            _state := 40;
        40:
            //            IF rfidInOut.stCompactModeInputMap.eResponseCode = _resetResponseCode THEN
            IF rfidInOut.xDone THEN
                THIS^.DoneWhen(TRUE);
                //                THIS^.Messenger.Info
                //                (
                //                    _stringbuilder.Append('Lock der Daten erfolgreich')
                //                        .Append('Startadresse: ')
                //                        .Append(TO_STRING(rfidinOut.udiStartAdress))
                //                        .Append(' Laenge: ')
                //                        .Append(TO_STRING(rfidInOut.uiDataLenght))
                //                        .ToString()
                //                );

                _state := 0;
            end_IF
    END_CASE
END_IF

{attribute 'monitoring' := 'call'}
PROPERTY ErrorId : RFID_FB_U.ERROR
GET
{warning disable C0371}
ErrorId := _eErrorID;
END_GET
END_PROPERTY

METHOD PUBLIC FB_init : BOOL
VAR_INPUT
    bInitRetains : BOOL; // if TRUE, the retain variables are initialized (warm start / cold start)
    bInCopyCode  : BOOL; // if TRUE, the instance afterwards gets moved into the copy code (online change)
    ParentObject : ITcoObject;
END_VAR
// This is not clear to me... I from time to time the consumer code does not see 'FB_init' of 'TcoObject', that's why overridden here with super call...
{warning disable C0316}
SUPER^.FB_init(bInitRetains, bInCopyCode, ParentObject);
END_METHOD

(*~
    <docu>
        <summary>
            Executes when task is aborted.
        </summary>
    </docu>
~*)
METHOD PROTECTED OnAbort
{warning disable C0371}
RfidInOut.eCommand := RFID_FB_U.COMMAND.IDLE;
RfidInOut.xExecute := FALSE;
RfidInOut.xAbort   := FALSE;
END_METHOD

(*~
    <docu>
        <summary>
            Executes when task reaches the ```Done``` state .
        </summary>
    </docu>
~*)
METHOD PROTECTED OnDone
{warning disable C0371}
rfidInOut.xExecute := FALSE;
rfidInOut.eCommand := RFID_FB_U.COMMAND.IDLE;
END_METHOD

(*~
    <docu>
        <summary>
            Executes when task reaches the ```Error``` state.
            <para>
                Do not confuse with <see cref="PlcDocu.TcoCore.TcoTask.WhileError()"/>, that is called cyclically until '''Error''' state is left.
            </para>
        </summary>
    </docu>
~*)
METHOD PROTECTED OnError
{warning disable C0371}
IF _noTagFound THEN
    _eErrorID := RFID_FB_U.ERROR.COMMAND_NO_TAG_FOUND;
    // not implemented by Turck
ELSIF rfidInOut.eErrorID = 16#2901 THEN
    _eErrorID := RFID_FB_U.ERROR.COMMAND_ADDRESS_OUTSIDE_BLOCK_BOUNDARIES;
ELSE
    _eErrorID := rfidInOut.eErrorID;
END_IF

THIS^.Messenger.Build().Append('Rfid Schreib/Lesekopf Fehler : ').Append(to_string(THIS^._eErrorID)).As().AsError();
END_METHOD

(*~
    <docu>
        <summary>
            Executes ones when the task starts (at the moment of transition from the ```Requested``` state into the ```Busy``` state).
        </summary>
    </docu>
~*)
METHOD PROTECTED OnStart
{warning disable C0371}
rfidInOut.eCommand := RFID_FB_U.COMMAND.IDLE;
rfidInOut.xExecute := FALSE;
rfidInOut.xAbort   := FALSE;
_state             := 10;
END_METHOD

(*~
    <docu>
        <summary>
            Restores this instance to the Ready state. Can be called explicitly or from within one of the restore mechanisms.
            <para>
                See also <see cref="PlcDocu.TcoCore.TcoTask.AutoRestorable()"/>
            </para>
        </summary>
    </docu>
~*)
METHOD Restore : ITcoRestorable
{warning disable C0371}
RfidInOut.eCommand := RFID_FB_U.COMMAND.IDLE;
RfidInOut.xExecute := FALSE;
RfidInOut.xAbort   := FALSE;
_noTagFound        := FALSE;
_eErrorID          := RFID_FB_U.ERROR.NO_ERROR;
SUPER^.Restore();
END_METHOD

END_FUNCTION_BLOCK

// ---- POUs/Turck Rfid Reader/Mock/RfidMockWorking.TcPOU
FUNCTION_BLOCK RfidMockWorking IMPLEMENTS IRfidHeadWrapper
VAR
    _timeOut        : Tc2_Standard.TON;
    _executionTimer : Tc2_Standard.TON := (PT := _executionTime);
    _executionTime  : TIME             := t#5ms;

    _udIntToMillis : UDINT := 1000;

    _resultUid : ARRAY[0..7] OF BYTE :=
    [
        16#E0
        , 16#04
        , 16#01
        , 16#50
        , 16#AC
        , 16#F4
        , 16#F3
        , 16#AD
    ];

    _states :
        (Idle
        , Busy
        , ElectedMethod
        , ReadUid
        , ReadData
        , WriteData
        , Error
        , Restore);
    _index : INT;

    _rfidInOut : RfidInOut;
END_VAR

{warning disable C0371}
//28 blocks, 4 bytes each, => 112 bytes max user Memory!

CASE _states OF
    Idle:
        _rfidInOut.xbusy := _rfidInOut.xExecute;
        _rfidInOut.xTP   := TRUE;

        IF _rfidInOut.xbusy THEN
            _states := Busy;
        END_IF

    Busy:

        _rfidInOut.uiDataRxLength := _rfidInOut.uiDataLenght;
        _timeOut(in := _rfidInOut.xbusy, PT := UDINT_TO_TIME(_rfidInOut.udiTimeOut) / _udintToMillis);
        _executionTimer(in := _rfidInOut.xBusy);

        IF _timeOut.Q THEN
            _states             := Error;
            _rfidInOut.eErrorID := RFID_FB_U.ERROR.TIME_OUT;
            RETURN;

        ELSIF _executionTimer.Q THEN
            _states := ElectedMethod;
        END_IF

    ElectedMethod:
        IF _rfidInOut.uiDataLenght > 112 THEN
            _states             := Error;
            _rfidInOut.eErrorID := RFID_FB_U.ERROR.COMMAND_LENGTH_OUTSIDE_TAG_SPECS;
            RETURN;
        ELSIF _rfidInOut.udiStartAdress > 112 THEN
            _states             := Error;
            _rfidInOut.eErrorID := RFID_FB_U.ERROR.COMMAND_ADDRESS_OUTSIDE_TAG_SPECS;
            RETURN;
        END_IF

        IF _rfidInOut.eCommand = RFID_FB_U.COMMAND.INVENTORY THEN
            FOR _index := 0 TO 7 DO
                _rfidInOut.myReadData[_index] := _resultUid[_index];
            END_FOR

            _rfidInOut.xbusy := FALSE;
            _rfidInOut.xDone := TRUE;
        ELSIF _rfidInOut.eCommand = RFID_FB_U.COMMAND.READ THEN

            FOR _index := 0 TO UINT_TO_INT(_rfidInOut.uiDataLenght) - 1 DO
                _rfidInOut.myReadData[_index] := 16#05 + INT_TO_BYTE(_index + UDINT_TO_INT(_rfidInOut.udiStartAdress));
            END_FOR

            _rfidInOut.xbusy := FALSE;
            _rfidInOut.xDone := TRUE; //

        ELSIF _rfidInOut.eCommand = RFID_FB_U.COMMAND.WRITE THEN
            _rfidInOut.xbusy := FALSE;
            _rfidInOut.xDone := TRUE;

        ELSIF _rfidInOut.eCommand = RFID_FB_U.COMMAND.SET_PERMA_LOCK THEN
            _rfidInOut.xbusy := FALSE;
            _rfidInOut.xDone := TRUE;
        END_IF

    Error:
        _executionTimer(in := FALSE);
        _timeOut(in := FALSE);
        _rfidInOut.xbusy  := FALSE;
        _rfidInOut.xError := TRUE;

        IF NOT _rfidInOut.xExecute THEN
            _States := Restore;
        END_IF
    Restore:
        _rfidInOut.xDone    := FALSE;
        _rfidInOut.xError   := FALSE;
        _rfidInOut.eErrorID := RFID_FB_U.ERROR.NO_ERROR;
        _States             := Idle;
END_CASE

METHOD Execute
VAR_INPUT
    xExecute       : BOOL;
    xAbort         : BOOL;
    udiTimeOut     : UDINT := 10000;
    eCommand       : RFID_FB_U.COMMAND;
    udiStartAdress : UDINT;
    uiDataLenght   : UINT;
    myWriteData    : ARRAY[0..127] OF BYTE;
END_VAR
VAR_OUTPUT
    myReadData          : ARRAY[0..127] OF BYTE;
    xDone               : BOOL;
    xBusy               : BOOL;
    xError              : BOOL;
    xAborted            : BOOL;
    eErrorID            : RFID_FB_U.ERROR;
    xTP                 : BOOL;
    xRWHeadNotCOnnected : BOOL;
    uiDataRxLength      : UINT;
END_VAR
VAR_INST
    _busy : BOOL;
END_VAR
THIS^();

_rfidInOut.xExecute       := xExecute;
_rfidInOut.xAbort         := xAbort;
_rfidInOut.udiTimeOut     := udiTimeOut;
_rfidInOut.eCommand       := eCommand;
_rfidInOut.udiStartAdress := udiStartAdress;
_rfidInOut.uiDataLenght   := uiDataLenght;
_rfidInOut.myWriteData    := myWriteData;

myReadData          := _rfidInOut.myReadData;
xDone               := _rfidInOut.xDone;
xBusy               := _rfidInOut.xBusy;
xError              := _rfidInOut.xError;
xAborted            := _rfidInOut.xAborted;
eErrorID            := _rfidInOut.eErrorID;
xTP                 := _rfidInOut.xTP;
xRWHeadNotCOnnected := _rfidInOut.xRWHeadNotCOnnected;
uiDataRxLength      := _rfidInOut.uiDataRxLength;
END_METHOD

END_FUNCTION_BLOCK

// ---- Test/Engel Ethercat Bridge Comm Tests/EngelInput_Test.TcPOU
FUNCTION_BLOCK EngelInput_Test EXTENDS TcUnit.FB_TestSuite
VAR

END_VAR

ParseVariantOne();

METHOD PRIVATE ParseVariantOne
VAR_INST
    in : ARRAY[1..42] OF BYTE;

    engelInput : EngelInput;

    inputData : EngelInputData;
END_VAR
// lebenssignal: alle 6ms muss der Zaehler um 1 erhoet werden (0-255, 0-255)
// will be the Counter be incremented from me and engel,
// will there be 2 Counter, everybody responsible for his
// what is the Result, if not incremented

//

Test('ParseVariantOne');

in[1]  := 255;
in[2]  := 255;
in[39] := 2#1111_1111;

engelInput(input := in);

inputData := engelInput.GetInputData();

AssertEquals_UINT(Expected := 65535, Actual := inputData.HeartBeat, 'Heartbeat not Correct');
AssertTrue(Condition := inputData.AutoActive, ' AutomatikActive should be true');
AssertTrue(Condition := inputData.HomeDone, 'HomeDoneshould be true');
AssertTrue(Condition := inputData.ManualActive, 'ManualActive should be true');
AssertTrue(Condition := inputData.HomeRequest, 'RequestHome should be true');
AssertTrue(Condition := inputData.SafetyClosed, 'SafetyClosed should be true');
AssertTrue(Condition := inputData.SafetyOpeningAllowed, 'SafetyOpeningAllowed should be true');
AssertTrue(Condition := inputData.AutoStart, 'StartAuto should be true');

TEST_FINISHED();
END_METHOD

END_FUNCTION_BLOCK

// ---- POUs/Engel Ethercat Bridge Communication/FunctionBlocks/EngelInput.TcPOU
FUNCTION_BLOCK EngelInput IMPLEMENTS IInput
VAR_INPUT
    input : ARRAY[1..42] OF BYTE;
END_VAR

METHOD GetInputData : EngelInputData
VAR
    hbTemp : uint;
END_VAR
hbTemp := input[1];
hbTemp := SHL(hbTemp, 8);
hbTemp := hbTemp OR input[2];

GetInputData.HeartBeat            := hbTemp;
GetInputData.ManualActive         := input[39].0;
GetInputData.AutoActive           := input[39].1;
GetInputData.AutoStart            := input[39].2;
GetInputData.HomeRequest          := input[39].3;
GetInputData.HomeDone             := input[39].4;
GetInputData.SafetyClosed         := input[39].5;
GetInputData.SafetyOpeningAllowed := input[39].6;
END_METHOD

END_FUNCTION_BLOCK

// ---- POUs/Engel Ethercat Bridge Communication/FunctionBlocks/HeartBeat.TcPOU
FUNCTION_BLOCK HeartBeat IMPLEMENTS IHeartBeat
VAR_INPUT
    execute : BOOL;
END_VAR

VAR
    heartBeatTimer : TON;
    eState         : eHeartBeatState;
    erroString     : T_MaxString;
    heartBeat      : UINT;

END_VAR

IF execute THEN
    heartBeatTimer();

    CASE eState OF
        eHeartBeatState.Unknown:
            CheckStates();
        eHeartBeatState.Valid:
            heartBeatTimer(in := TRUE);
            erroString := '';
            CheckStates();
        eHeartBeatState.Timeout:
            erroString := CONCAT
            (
                'Timeout, da keine Erhoehung Heartbeat stattgefunden hat in '
                , TO_STRING(GetHeartBeatTimeOutTime)
            );
    ELSE
        ;
    END_CASE
END_IF

METHOD PRIVATE CheckStates : BOOL
VAR_INPUT
END_VAR
IF execute THEN
    IF heartBeatTimer.Q THEN
        SetState(eHeartBeatState.Timeout);
    END_IF
ELSE
    SetState(eHeartBeatState.Unknown);
END_IF
END_METHOD

METHOD FB_init : BOOL
VAR_INPUT
    bInitRetains         : BOOL; // if TRUE, the retain variables are initialized (warm start / cold start)
    bInCopyCode          : BOOL; // if TRUE, the instance afterwards gets moved into the copy code (online change)
    heartBeatTimeoutTime : TIME;
END_VAR
heartBeatTimer.PT := heartBeatTimeoutTime;

this^.eState := eHeartBeatState.Unknown;
END_METHOD

PROPERTY GetErrorMessage : T_MaxString;
GET
GetErrorMessage := erroString;
END_GET
END_PROPERTY

//actual Heartbeat of PLC
PROPERTY GetHeartBeat : UINT
GET
IF NOT execute THEN
    THIS^.erroString := 'Bitte Execute auf True setzten!';
    RETURN;
END_IF

GetHeartBeat := heartBeat;
END_GET
END_PROPERTY

PROPERTY GetHeartbeatTimeoutTime : TIME
GET
GetHeartbeatTimeoutTime := heartBeatTimer.PT;
END_GET
END_PROPERTY

PROPERTY GetState : eHeartBeatState
GET
GetState := eState;
END_GET
END_PROPERTY

// Increases HB +1 from InputValue
METHOD IncreaseHeartBeat : UINT
VAR_INPUT
    externalHeartBeat : UINT;
END_VAR
IF NOT execute THEN
    THIS^.erroString  := 'Bitte Execute auf True setzten!';
    IncreaseHeartBeat := 0;
    RETURN;
END_IF

SetState(eHeartBeatState.Valid);
ResetTimer();

IF externalHeartBeat >= 255 THEN
    IncreaseHeartBeat := 0;
ELSE
    IncreaseHeartBeat := externalHeartBeat + 1;
END_IF

heartBeat := IncreaseHeartBeat;
END_METHOD

METHOD PRIVATE ResetTimer
VAR_INPUT
END_VAR
THIS^.heartBeatTimer(IN := false);
END_METHOD

METHOD PRIVATE SetState
VAR_INPUT
    eState : eHeartBeatState;
END_VAR
This^.eState := eState;
END_METHOD

END_FUNCTION_BLOCK

// ---- Test/Engel Ethercat Bridge Comm Tests/EngelOutput_Test.TcPOU
FUNCTION_BLOCK EngelOutput_Test EXTENDS FB_TestSuite

SetOutputsAndVerify();

METHOD PRIVATE SetOutputsAndVerify
VAR
    out : EngelOutput;
END_VAR
TEST('SetOutputsAndVerify');

out.ManualActive(TRUE);
AssertEquals_BYTE(Expected := 2#0000_0001, Actual := out.output[39], 'SetManualActive is true');
out.ManualActive(FALSE);

out.AutomaticIsActive(TRUE);
AssertEquals_BYTE(Expected := 2#0000_0010, Actual := out.output[39], 'SetAutomaticeActive is true');
out.AutomaticIsActive(FALSE);

out.StartAutomatic(TRUE);
AssertEquals_BYTE(Expected := 2#0000_0100, Actual := out.output[39], 'SetStart is true');
out.StartAutomatic(FALSE);

out.RequestHome(TRUE);
AssertEquals_BYTE(Expected := 2#0000_1000, Actual := out.output[39], 'SetRequestHome is true');
out.RequestHome(FALSE);

out.HomeIsDone(TRUE);
AssertEquals_BYTE(Expected := 2#0001_0000, Actual := out.output[39], 'SetHomeDone is true');
out.HomeIsDone(FALSE);

out.SafetyIsClosed(TRUE);
AssertEquals_BYTE(Expected := 2#0010_0000, Actual := out.output[39], 'SetSafetyClosed is true');
out.SafetyIsClosed(FALSE);

out.RequestSafetyOpening(TRUE);
AssertEquals_BYTE(Expected := 2#0100_0000, Actual := out.output[39], 'SetSafetyOpeningRequest is true');
out.RequestSafetyOpening(FALSE);

out.SetHeartBeat(65535);
AssertEquals_BYTE(Expected := 255, Actual := out.output[1], 'Byte  1 Heartbeat shall be 255');
AssertEquals_BYTE(Expected := 255, Actual := out.output[2], 'Byte  2 Heartbeat shall be 255');

TEST_FINISHED();
END_METHOD

END_FUNCTION_BLOCK

// ---- POUs/Engel Ethercat Bridge Communication/FunctionBlocks/EngelOutput.TcPOU
FUNCTION_BLOCK EngelOutput IMPLEMENTS IOutput
VAR_OUTPUT
    output : ARRAY[0..42] OF BYTE;
END_VAR

METHOD PUBLIC AutomaticIsActive
VAR_INPUT
    enable : BOOL;
END_VAR

output[39].1 := enable;
END_METHOD

METHOD PUBLIC HomeIsDone
VAR_INPUT
    enable : BOOL;
END_VAR
output[39].4 := enable;
END_METHOD

METHOD PUBLIC ManualActive
VAR_INPUT
    enable : BOOL;
END_VAR
output[39].0 := enable;
END_METHOD

METHOD PUBLIC RequestHome
VAR_INPUT
    enable : BOOL;
END_VAR
output[39].3 := enable;
END_METHOD

METHOD PUBLIC RequestSafetyOpening
VAR_INPUT
    enable : BOOL;
END_VAR
output[39].6 := enable;
END_METHOD

METHOD PUBLIC SafetyIsClosed
VAR_INPUT
    enable : BOOL;
END_VAR
output[39].5 := enable;
END_METHOD

METHOD SetHeartBeat
VAR_INPUT
    heartBeat : UINT;
END_VAR
output[1].0 := heartBeat.0;
output[1].1 := heartBeat.1;
output[1].2 := heartBeat.2;
output[1].3 := heartBeat.3;
output[1].4 := heartBeat.4;
output[1].5 := heartBeat.5;
output[1].6 := heartBeat.6;
output[1].7 := heartBeat.7;

output[2].0 := heartBeat.8;
output[2].1 := heartBeat.9;
output[2].2 := heartBeat.10;
output[2].3 := heartBeat.11;
output[2].4 := heartBeat.12;
output[2].5 := heartBeat.13;
output[2].6 := heartBeat.14;
output[2].7 := heartBeat.15;
END_METHOD

METHOD PUBLIC StartAutomatic
VAR_INPUT
    enable : BOOL;
END_VAR
output[39].2 := enable;
END_METHOD

END_FUNCTION_BLOCK

// ---- Test/Engel Ethercat Bridge Comm Tests/HeartBeat_Test.TcPOU
FUNCTION_BLOCK HeartBeat_Test EXTENDS TcUnit.FB_TestSuite

GetsValueAndGiveBackIncreasedValueStatusValid();
HeartbeatFromEngelTimeout_GetStateGivesStatusTimeOut();
ErrorOccurs_ExpectStringMessage();
AfterTimeOutRecieveNewHb_ExpectToChangeStatusBackToValid();
NotExecute_ExpectErrorMessageAndStateUnknown();

METHOD PRIVATE AfterTimeOutRecieveNewHb_ExpectToChangeStatusBackToValid
VAR_INST
    toTimer : TON := (PT := T#4MS); // Bigger 12ms !
    eState  : eHeartBeatState;
    first   : BOOL := TRUE;
    hb      : HeartBeat(heartBeatTimeoutTime := T#2MS);
    resetHb : BOOL;

END_VAR
Test('ErrorOccurs_ExpectStringAfterTimeOutRecieveNewHb_ExpectToChangeStatusBackToValidMessage');
// Arrange
// Act
// Assert
hb(execute := TRUE);
toTimer();

IF first THEN
    first  := FALSE;
    eState := hb.GetState;
    hb.IncreaseHeartBeat(5);
    eState := hb.GetState;
    AssertEquals_UINT(6, hb.GetHeartBeat, 'Nach Erhoehung muss HB 6 sein');
    AssertTrue(eState = eHeartBeatState.Valid, 'State muss Valid sein');
    toTimer(in := TRUE);
END_IF

IF toTimer.q THEN
    AssertTrue(hb.GetState = eHeartBeatState.Timeout, 'Timeout, keine Erhoehung HB durch Engel');
    resetHb := TRUE;
END_IF

IF resetHb THEN
    hb.IncreaseHeartBeat(665);
    AssertTrue(hb.GetState = eHeartBeatState.Valid, 'State muss Valid sein');
    AssertEquals_UINT(0, hb.GetHeartBeat, 'Nach Erhoehung muss HB 0 sein');

    TEST_FINISHED();
END_IF
END_METHOD

METHOD PRIVATE ErrorOccurs_ExpectStringMessage
VAR_INST
    hb                 : HeartBeat(heartBeatTimeoutTime := T#1MS);
    toTimer            : TON := (PT := T#3MS); // Bigger 12ms !
    errorMessage       : STRING;
    actualErrorMessage : STRING;
    first              : BOOL := TRUE;
    eState             : eHeartBeatState;

END_VAR
Test('ErrorOccurs_ExpectStringMessage');
// Arrange
// Act
// Assert

hb(execute := TRUE);
toTimer(in := TRUE);

IF first THEN
    errorMessage       := '';
    actualErrorMessage := hb.GetErrorMessage;
    AssertEquals_STRING(errorMessage, actualErrorMessage, 'ErrorMessage soll leer sein');
    first := FALSE;
    hb.IncreaseHeartBeat(1);
END_IF

IF toTimer.Q THEN
    eState := hb.GetState;
    AssertTrue(eState = eHeartBeatState.Timeout, 'Timeout, keine Erhoehung HB durch Engel');
    actualErrorMessage := hb.GetErrorMessage;

    errorMessage := CONCAT
    (
        'Timeout, da keine Erhoehung Heartbeat stattgefunden hat in '
        , TO_STRING(hb.GetHeartBeatTimeOutTime)
    );

    AssertEquals_STRING(errorMessage, actualErrorMessage, 'ErrorMessage muss gleich sein');

    TEST_FINISHED();
end_if
END_METHOD

METHOD PRIVATE GetsValueAndGiveBackIncreasedValueStatusValid
VAR
    hb            : HeartBeat(heartBeatTimeoutTime := T#12MS);
    eState        : eHeartBeatState;
    inputData     : UINT;
    inHeartBeat   : UINT := 0;
    expectedOutHb : UINT := 1;
END_VAR
// Calculate a Heartbeat for the Engle Ethercat Bridge Communication
// Wertebereich des Heartbeats ist [0..65635]
// Aber Engel erhoeht internen Zaehler alle 6ms bis 255!
// Nur Aenderung von meiner Seite notwendig
// Wenn nach max. 12ms keine Aenderung => Fehler

Test('GetsValueAndGiveBackIncreasedValueStatusValid');
// Arrange
// Act
// Assert

hb(execute := TRUE);

eState := hb.GetState;
AssertTrue(estate = eHeartBeatState.Unknown, 'State soll Unknown sein');
///=========================================================

inputData := hb.IncreaseHeartBeat(inHeartBeat);
eState    := hb.GetState;
AssertEquals_UINT(expectedOutHb, inputData, 'Nach Erhoehung muss HB 1 sein');
AssertTrue(estate = eHeartBeatState.Valid, 'State muss Valid sein');

//Arrange
inHeartBeat   := 255;
expectedOutHb := 0;

//Act
inputData := hb.IncreaseHeartBeat(inHeartBeat);
AssertEquals_UINT(expectedOutHb, inputData, 'Nach Erhoehung ueber 255 muss HB wieder 0 sein');
AssertTrue(estate = eHeartBeatState.Valid, 'State muss Valid sein');

TEST_FINISHED();
END_METHOD

METHOD PRIVATE HeartbeatFromEngelTimeout_GetStateGivesStatusTimeOut
VAR
    inputData     : UINT;
    inHeartBeat   : UINT := 22;
    expectedOutHb : UINT := 23;
END_VAR

VAR_INST
    toTimer : TON := (PT := T#20MS); // Bigger 12ms !
    eState  : eHeartBeatState;
    first   : BOOL := TRUE;
    hb      : HeartBeat(heartBeatTimeoutTime := T#12MS);

END_VAR
// Calculate a Heartbeat for the Engle Ethercat Bridge Communication
// Wertebereich des Heartbeats ist [0..65635]
// Aber Engel erhoeht internen Zaehler alle 6ms bis 255!
// Nur Aenderung von meiner Seite notwendig
// Wenn nach max. 12ms keine Aenderung => Fehler

Test('HeartbeatFromEngelTimeout_GetStateGivesStatusTimeOut');
// Arrange
// Act
// Assert
hb(execute := TRUE);
toTimer();

IF first THEN
    first  := FALSE;
    eState := hb.GetState;
    AssertTrue(estate = eHeartBeatState.Unknown, 'State soll Unknown sein');
    ///=========================================================

    inputData := hb.IncreaseHeartBeat(inHeartBeat);
    eState    := hb.GetState;
    AssertEquals_UINT(expectedOutHb, inputData, 'Nach Erhoehung muss HB 23 sein');
    AssertEquals_UINT(expectedOutHb, hb.GetHeartBeat, 'Bie GetHeartBeat muss HB 23 sein');
    AssertTrue(estate = eHeartBeatState.Valid, 'State muss Valid sein');
    //======================

    toTimer(in := TRUE);
END_IF

IF toTimer.ET <= T#12MS THEN
    AssertTrue(estate = eHeartBeatState.Valid, 'Valid, TO erst nach 12ms');
END_IF

IF toTimer.Q THEN
    eState := hb.GetState;
    AssertTrue(estate = eState, 'Timeout, keine Erhoehung HB durch Engel');
    TEST_FINISHED();
END_IF
END_METHOD

METHOD PRIVATE NotExecute_ExpectErrorMessageAndStateUnknown
VAR
    timeout             : TIME := T#1MS;
    hb                  : HeartBeat(heartBeatTimeoutTime := timeout);
    errorStringExpected : STRING;
    errorStringActual   : STRING;
END_VAR
TEST('NotExecute_ExpectErrorMessageAndStateUnknown');

hb(execute := FALSE);
hb.IncreaseHeartBeat(23);
errorStringExpected := 'Bitte Execute auf True setzten!';
errorStringActual   := hb.GetErrorMessage;
AssertEquals_STRING(errorStringActual, errorStringExpected, 'ErrorMessage soll gleich sein');
AssertTrue(hb.GetState = eHeartBeatState.Unknown, 'State muss Unknown sein');
AssertEquals_UINT(hb.IncreaseHeartBeat(25), 0, 'Keine Erhoehung, da Execute False');
AssertEquals_UINT(hb.GetHeartBeat, 0, 'Keine Erhoehung, da Execute False');
AssertTrue(hb.GetHeartbeatTimeoutTime = timeout, 'Property muss gleiche Zeit wie bei Init zurueckgeben (1ms)');

TEST_FINISHED();
END_METHOD

END_FUNCTION_BLOCK

// ---- Test/Sequences/Test/SequenceTryout_Test.TcPOU
FUNCTION_BLOCK SequenceTryout_Test EXTENDS TcUnit.FB_TestSuite IMPLEMENTS TcoCore.ITcoContext
VAR
    //Context for TcOpen
    _nfContext : TcoCore.TcoContextNfCompatibility;
END_VAR

VAR
    //~
    autoSequenceTryOutTest : SequenceTryout(THIS^, eRestoreMode.AutoRestoreMembers);
    //~
END_VAR


_nfContext.VolatileOpen(); //Required for TCopen
//==============================================
GivenThatEverythingWorksExpectCompleteSequenceToFinishInDone();
//==============================================
_nfContext.VolatileClose();

PROPERTY Context : TcoCore.ITcoContext
GET
Context := This^._nfContext;
END_GET
END_PROPERTY

PROPERTY EndCycleCount : ULINT
GET
EndCycleCount := THIS^._nfContext._endCycleCount;
END_GET
END_PROPERTY

PROPERTY Environment : TcoCore.ITcoContextEnvironment
GET
Environment := THIS^._nfContext._settings;
END_GET
END_PROPERTY

METHOD PRIVATE GivenThatEverythingWorksExpectCompleteSequenceToFinishInDone

VAR
    state                : INT;
    context              : ITcoContext;
    autoRestorable       : BOOL;
    currentStep          : StepDetails;
    euqalsTo             : BOOL;
    identity             : ULINT;
    isAutoRestoreEnabled : BOOL;
    isFreshState         : BOOL;
    lastStateChangeCycle : ULINT;
    messenger            : ITcoMessenger;
    modeController       : ITcoSequencerModeController;
    observer             : ITcoSequencerObserver;
    parent               : ITcoObject;

END_VAR

VAR
    currentStepActive : StepDetails;
END_VAR
//{warning disable C0371}
TcUnit.TEST('GivenThatEverythingWorksExpectCompleteSequenceToFinishInDone');
//Arrange

//autoSequenceTryOutTest.Restore();
currentStepActive.ID := 0;

////Act
autoSequenceTryOutTest.Run();

////Assert

//AssertEquals(Expected := currentStepActive.ID, Actual := autoSequenceTryOutTest.CurrentStep.ID, Message := 'Muss Step 999 sein');

state                := autoSequenceTryOutTest.State;
context              := autoSequenceTryOutTest.Context;
autorestorable       := autoSequenceTryOutTest.AutoRestorable;
currentStep          := autoSequenceTryOutTest.CurrentStep;
Identity             := autoSequenceTryOutTest.Identity;
isAutoRestoreEnabled := autoSequenceTryOutTest.IsAutoRestoreEnabled;
isFreshState         := autoSequenceTryOutTest.IsFreshState;
LastStateChangeCycle := autoSequenceTryOutTest.LastStateChangeCycle;
messenger            := autoSequenceTryOutTest.Messenger;
ModeController       := autoSequenceTryOutTest.ModeController;
Observer             := autoSequenceTryOutTest.Observer;
Parent               := autoSequenceTryOutTest.Parent;

IF (autoSequenceTryOutTest.CurrentStep.Duration >= T#10MS) OR autoSequenceTryOutTest.State = 999 THEN
    //autoSequenceTryOutTest.Restore();
    currentStepActive.ID := 999;
    AssertEquals
    (
        Expected  := currentStepActive.ID
        , Actual  := autoSequenceTryOutTest.CurrentStep.ID
        , Message := 'Muss Step 999 sein'
    );

    TcUnit.TEST_FINISHED();
END_IF
END_METHOD

PROPERTY Identity : ULINT
GET
Identity := THIS^._nfContext._Identity;
END_GET
END_PROPERTY

PROPERTY Logger : TcoCore.ITcoLogger
GET
Logger := THIS^._nfContext._logger;
END_GET
END_PROPERTY

PROPERTY RealTimeClock : TcoCore.ITcoRtc
GET
RealTimeClock := THIS^._nfContext._rtc;
END_GET
END_PROPERTY

PROPERTY StartCycleCount : ULINT
GET
StartCycleCount := THIS^._nfContext._startCycleCount;
END_GET
END_PROPERTY

END_FUNCTION_BLOCK

// ---- POUs/Sequences/Test/SequenceTryout.TcPOU
FUNCTION_BLOCK SequenceTryout EXTENDS TcoCore.TcoSequencer
VAR
    counter : INT;
END_VAR
VAR
    //    eSequenceTest : E_SequenceTest := E_SequenceTest.WaitForStart;
    eSequenceTest : stSequenceTest;
    itfValveA     : I_DualPositionActuator := valveA;
    //~
    valveA : FB_DualPositionActuator
    (
        tActivateTimeout                     := T#3S
        , tDisableTimeout                    := T#3S
        , bIsActiveFeedbackSensorAvailable   := TRUE
        , bIsDisabledFeedbackSensorAvailable := TRUE
        , bNormallyDisabled                  := TRUE
    );
    //~
END_VAR
VAR CONSTANT
    simV : INT := 4;
END_VAR

(*~
    <docu>
        <summary>
            Main method of the sequener. Custom code needs to be placed here. The sequencer is executed by call of InstanceName.Run() method.
            This method is abstract, and it must be overridden in derived block.
        </summary>
    </docu>
~*)
METHOD PROTECTED Main : BOOL
counter := counter + 1;

IF (Step(eSequenceTest.WaitForStart, TRUE, 'Restore und Start')) THEN
    //    eSequenceTest := stSequenceTest.OpenValveAandB;
    StepCompleteWhen(counter MOD simV = 0);
END_IF

IF (Step(eSequenceTest.OpenValveAandB, TRUE, 'Zweiter Step')) THEN
    StepCompleteWhen(counter MOD simV = 0);
END_IF

IF (Step(999, TRUE, 'SEQUENCE COMPLETE')) THEN
    //--------------------------------------------
    CompleteSequence();
    //--------------------------------------------
END_IF;

IF (step(909, TRUE, 'ERROR Handling')) THEN
    ;
END_IF
END_METHOD

(*~
    <docu>
        <summary>
            This method is executed upon step completion.
            This method can be overridden in derived block by custom logic.
        </summary>
    </docu>
~*)
METHOD PROTECTED OnStepCompleted
counter := 1;
END_METHOD

END_FUNCTION_BLOCK

// ---- POUs/Counter Allgemein/Counter.TcPOU
//{attribute 'hide_all_locals'}
FUNCTION_BLOCK Counter EXTENDS TcoCore.TcoObject IMPLEMENTS ICounter
VAR
    _countStep  : UDINT;
    _countValue : UDINT;
    _countLimit : UDINT;

END_VAR

METHOD CountDown
_countValue := _countValue - _countStep;
END_METHOD

{attribute 'monitoring' := 'variable'}
PROPERTY CountLimitReached : BOOL
GET
CountLimitReached := CountValue >= _countLimit;
END_GET
END_PROPERTY

METHOD CountUp

_countValue := _countValue + _countStep;
END_METHOD

{attribute 'monitoring' := 'monitor'}
PROPERTY CountValue : UDINT
GET
CountValue := _countValue;
END_GET
END_PROPERTY

{attribute 'monitoring' := 'variable'}
PROPERTY CountZeroReached : BOOL
GET
CountZeroReached:= CountValue = 0;
END_GET
END_PROPERTY

{attribute 'hide'}
METHOD FB_init : BOOL
VAR_INPUT
    (* if TRUE, the retain variables are initialized (warm start / cold start)*)
    bInitRetains : BOOL;
    (* if TRUE, the instance afterwards gets moved into the copy code (online change)*)
    bInCopyCode  : BOOL;
    ParentObject : ITcoObject;

    countStep      : UDINT;
    countInitValue : UDINT;
    countLimit     : UDINT;
END_VAR
//SUPER^.FB_init(bInitRetains, bInCopyCode, ParentObject);

_countStep := countStep;
_countValue := countInitValue;
_countLimit := countLimit;

IF countInitValue > countLimit THEN
    Messenger.Error('Value groesser als Limit eingestellt');
    RETURN;
END_IF
END_METHOD

METHOD ResetCount
_countValue := 0;
END_METHOD

END_FUNCTION_BLOCK

// ---- POUs/DualPositionActuator/POUs/FB_DualPositionActuator.TcPOU
FUNCTION_BLOCK FB_DualPositionActuator IMPLEMENTS I_DualPositionActuator
VAR
    {attribute 'TcHmiSymbol.Show'}
    {attribute 'TcHmiSymbol.ReadOnly'}
    eState                             : E_DualPositionActuatorState;
    fbTimerActivatingTimeout           : TON;
    fbTimerDisablingTimeout            : TON;
    bIsActiveFeedbackSensorAvailable   : BOOL;
    bIsDisabledFeedbackSensorAvailable : BOOL;

    bIsNormallyDisabled : BOOL; // [True = Normally disabled, False = Normally activated]
END_VAR
VAR_INPUT
    bActiveFeedback  : BOOL; // Sensor input
    bDisableFeedback : BOOL; // Sensor input
END_VAR
VAR_OUTPUT
    bActivate : BOOL; // Actuator output
    bDisable  : BOOL; // Actuator output
END_VAR

CASE eState OF
    E_DualPositionActuatorState.Unknown:
        CheckFeedback();

    E_DualPositionActuatorState.Active:
        CheckFeedback();

    E_DualPositionActuatorState.Disabled:
        CheckFeedback();

    E_DualPositionActuatorState.TimeoutActivating:
        IF bIsNormallyDisabled THEN
            bActivate := FALSE;
        ELSE
            CheckFeedback();
        END_IF

    E_DualPositionActuatorState.TimeoutDisabling:
        IF NOT bIsNormallyDisabled THEN
            bDisable := FALSE;
        ELSE
            CheckFeedback();
        END_IF

    E_DualPositionActuatorState.Activating:
        IF NOT bIsActiveFeedbackSensorAvailable AND NOT bIsDisabledFeedbackSensorAvailable THEN
            SetState(eState := E_DualPositionActuatorState.Active);
        ELSIF NOT bIsActiveFeedbackSensorAvailable AND NOT bDisableFeedback THEN
            SetState(eState := E_DualPositionActuatorState.Active);
        ELSIF NOT bIsActiveFeedbackSensorAvailable AND bDisableFeedback THEN
            fbTimerActivatingTimeout(IN := TRUE);

            IF fbTimerActivatingTimeout.Q THEN
                SetState(eState := E_DualPositionActuatorState.TimeoutActivating);
            END_IF
        ELSE
            fbTimerActivatingTimeout(IN := TRUE);

            IF fbTimerActivatingTimeout.Q THEN
                SetState(eState := E_DualPositionActuatorState.TimeoutActivating);
            END_IF

            CheckFeedback();
        END_IF

    E_DualPositionActuatorState.Disabling:
        IF NOT bIsDisabledFeedbackSensorAvailable AND NOT bIsActiveFeedbackSensorAvailable THEN
            SetState(eState := E_DualPositionActuatorState.Disabled);
        ELSIF NOT bIsDisabledFeedbackSensorAvailable AND NOT bActiveFeedback THEN
            SetState(eState := E_DualPositionActuatorState.Disabled);
        ELSIF NOT bIsDisabledFeedbackSensorAvailable AND bActiveFeedback THEN
            fbTimerDisablingTimeout(IN := TRUE);

            IF fbTimerDisablingTimeout.Q THEN
                SetState(eState := E_DualPositionActuatorState.TimeoutDisabling);
            END_IF
        ELSE
            fbTimerDisablingTimeout(IN := TRUE);

            IF fbTimerDisablingTimeout.Q THEN
                SetState(eState := E_DualPositionActuatorState.TimeoutDisabling);
            END_IF

            CheckFeedback();
        END_IF
END_CASE

METHOD PUBLIC Activate
IF GetState() = E_DualPositionActuatorState.Activating OR GetState() = E_DualPositionActuatorState.Active THEN
    RETURN;
END_IF

SetState(eState := E_DualPositionActuatorState.Activating);
fbTimerActivatingTimeout(IN := FALSE);
bDisable  := FALSE;
bActivate := TRUE;
END_METHOD

METHOD PRIVATE CheckFeedback
IF eState = E_DualPositionActuatorState.TimeoutActivating OR eState = E_DualPositionActuatorState.TimeoutDisabling THEN
    RETURN;
ELSIF bActiveFeedback AND NOT bDisableFeedback AND eState <> E_DualPositionActuatorState.Disabling THEN
    SetState(eState := E_DualPositionActuatorState.Active);
ELSIF bDisableFeedback AND NOT bActiveFeedback AND eState <> E_DualPositionActuatorState.Activating THEN
    SetState(eState := E_DualPositionActuatorState.Disabled);
ELSIF NOT bActiveFeedback
          AND bIsActiveFeedbackSensorAvailable
          AND NOT bIsDisabledFeedbackSensorAvailable
          AND eState <> E_DualPositionActuatorState.Activating THEN
    SetState(eState := E_DualPositionActuatorState.Disabled);
ELSIF NOT bDisableFeedback
          AND bIsDisabledFeedbackSensorAvailable
          AND NOT bIsActiveFeedbackSensorAvailable
          AND eState <> E_DualPositionActuatorState.Disabling THEN
    SetState(eState := E_DualPositionActuatorState.Active);
ELSIF bActiveFeedback AND bDisableFeedback THEN
    SetState(eState := E_DualPositionActuatorState.Unknown);
END_IF
END_METHOD

METHOD PUBLIC Disable
IF GetState() = E_DualPositionActuatorState.Disabling OR GetState() = E_DualPositionActuatorState.Disabled THEN
    RETURN;
END_IF

SetState(eState := E_DualPositionActuatorState.Disabling);
fbTimerDisablingTimeout(IN := FALSE);
bDisable  := TRUE;
bActivate := FALSE;
END_METHOD

METHOD FB_init : BOOL
VAR_INPUT
    bInitRetains     : BOOL; // if TRUE, the retain variables are initialized (warm start / cold start)
    bInCopyCode      : BOOL; // if TRUE, the instance afterwards gets moved into the copy code (online change)
    tActivateTimeout : TIME;
    tDisableTimeout  : TIME;
    bIsActiveFeedbackSensorAvailable
        : BOOL;                                // Set this to true if feedback is provided by a sensor
    bIsDisabledFeedbackSensorAvailable : BOOL; // Set this to true if feedback is provided by a sensor
    bNormallyDisabled                  : BOOL; // [True = Normally disabled, False = Normally activated]
END_VAR
fbTimerActivatingTimeout.PT := tActivateTimeout;
fbTimerDisablingTimeout.PT  := tDisableTimeout;

THIS^.bIsActiveFeedbackSensorAvailable   := bIsActiveFeedbackSensorAvailable;
THIS^.bIsDisabledFeedbackSensorAvailable := bIsDisabledFeedbackSensorAvailable;

IF bNormallyDisabled AND NOT bIsDisabledFeedbackSensorAvailable THEN
    SetState(eState := E_DualPositionActuatorState.Disabled);
ELSIF NOT bNormallyDisabled AND NOT bIsActiveFeedbackSensorAvailable THEN
    SetState(eState := E_DualPositionActuatorState.Active);
END_IF

THIS^.bIsNormallyDisabled := bNormallyDisabled;
END_METHOD

METHOD GetDisableTimeoutTime : TIME
GetDisableTimeoutTime := fbTimerDisablingTimeout.PT;
END_METHOD

METHOD GetEnableTimeoutTime : TIME
GetEnableTimeoutTime := fbTimerActivatingTimeout.PT;
END_METHOD

METHOD PUBLIC GetState : E_DualPositionActuatorState
GetState := THIS^.eState;
END_METHOD

METHOD SetDisableTimeoutTime
VAR_INPUT
    tDisableTimeoutTime : TIME;
END_VAR
fbTimerDisablingTimeout.PT := tDisableTimeoutTime;
END_METHOD

METHOD SetEnableTimeoutTime
VAR_INPUT
    tEnableTimeoutTime : TIME;
END_VAR
fbTimerActivatingTimeout.PT := tEnableTimeoutTime;
END_METHOD

METHOD PRIVATE SetState
VAR_INPUT
    eState : E_DualPositionActuatorState;
END_VAR
THIS^.eState := eState;
END_METHOD

END_FUNCTION_BLOCK

// ---- Test/DualPositionActuator/FB_DualPositionActuator_Test.TcPOU
FUNCTION_BLOCK FB_DualPositionActuator_Test EXTENDS TcUnit.FB_TestSuite
VAR

END_VAR

ActiveFeedbackSensorAvailableButNotDisableFeedbackAvailableIfNoActiveFeedbackProvidedItShouldGoToDisabled();
BothSensorInputsAreTrueExpectUnknownState();
CloseOneSensorActuatorExpectItToBeClosedWithoutFeedback();
CloseOneSensorActuatorExpectItToBeClosedWithoutFeedbackVariant2();
CloseOneSensorActuatorExpectItToTimeout();
CloseTwoSensorActuatorExpectCloseOutputToBeTrue();
CloseTwoSensorActuatorExpectItToBeClosed();
CloseTwoSensorActuatorExpectItToTimeout();
DisableFeedbackSensorAvailableButNotActiveFeedbackAvailableIfNoDisableFeedbackProvidedItShouldGoToActive();
DisableTwoSensorNormallyEnabledActuatorExpectItToTimeoutThenExpectDisablingToGoLow();
EnableTwoSensorNormallyDisabledActuatorExpectItToTimeoutThenExpectActuationToGoLow();
GivenActivatedFeedBackSensorNotAvailableAndNormallyActivatedThenShouldBeActivated();
GivenDisabledFeedBackSensorNotAvailableAndNormallyDisabledThenShouldBeDisabled();
OpenOneSensorActuatorExpectItToBeOpenWithoutFeedback();
OpenOneSensorActuatorExpectItToBeOpenWithoutFeedbackVariant2();
OpenOneSensorActuatorExpectItToTimeout();
OpenTwoSensorActuatorExpectItToBeOpen();
OpenTwoSensorActuatorExpectItToTimeout();

METHOD PRIVATE
    ActiveFeedbackSensorAvailableButNotDisableFeedbackAvailableIfNoActiveFeedbackProvidedItShouldGoToDisabled
VAR_INST
    fbActuator : FB_DualPositionActuator
    (
        tActivateTimeout                     := T#5MS
        , tDisableTimeout                    := T#5MS
        , bIsActiveFeedbackSensorAvailable   := TRUE
        , bIsDisabledFeedbackSensorAvailable := FALSE
        , bNormallyDisabled                  := TRUE
    );
    nTestState : INT;
END_VAR
TEST('ActiveFeedbackSensorAvailableButNotDisableFeedbackAvailableIfNoActiveFeedbackProvidedItShouldGoToDisabled');

CASE nTestState OF
    0:
        fbActuator(bActiveFeedback := TRUE);
        AssertEquals_INT
        (
            Expected  := E_DualPositionActuatorState.Active
            , Actual  := fbActuator.GetState()
            , Message := 'Actuator should be active'
        );

        nTestState := nTestState + 1;

    1:
        fbActuator(bActiveFeedback := FALSE);
        AssertEquals_INT
        (
            Expected  := E_DualPositionActuatorState.Disabled
            , Actual  := fbActuator.GetState()
            , Message := 'Actuator should be disabled'
        );

        nTestState := nTestState + 1;
    2:
        {analysis -9}
        TEST_FINISHED();
END_CASE
END_METHOD

METHOD PRIVATE BothSensorInputsAreTrueExpectUnknownState
VAR
    fbActuator : FB_DualPositionActuator
    (
        tActivateTimeout                     := T#10MS
        , tDisableTimeout                    := T#10MS
        , bIsActiveFeedbackSensorAvailable   := TRUE
        , bIsDisabledFeedbackSensorAvailable := TRUE
        , bNormallyDisabled                  := TRUE
    );
END_VAR
TEST('BothSensorInputsAreTrueExpectUnknownState');

fbActuator(bActiveFeedback := TRUE, bDisableFeedback := TRUE);

AssertTrue(Condition := fbActuator.GetState() = E_DualPositionActuatorState.Unknown, Message := '');

{analysis -9}
TEST_FINISHED();
END_METHOD

METHOD PRIVATE CloseOneSensorActuatorExpectItToBeClosedWithoutFeedback
VAR_INST
    fbActuator : FB_DualPositionActuator
    (
        tActivateTimeout                     := T#5MS
        , tDisableTimeout                    := T#5MS
        , bIsActiveFeedbackSensorAvailable   := TRUE
        , bIsDisabledFeedbackSensorAvailable := FALSE
        , bNormallyDisabled                  := TRUE
    );

    fbTestTimer : TON := (PT := T#2MS);
    bRunOnce    : BOOL;
END_VAR
TEST('CloseOneSensorActuatorExpectItToBeClosedWithoutFeedback');
fbTestTimer(IN := TRUE);

IF NOT bRunOnce THEN
    bRunOnce := TRUE;
    fbActuator.Disable();
END_IF

fbActuator(bActiveFeedback := FALSE, bDisableFeedback := FALSE);

IF fbTestTimer.Q THEN
    AssertEquals_INT
    (
        Expected  := E_DualPositionActuatorState.Disabled
        , Actual  := fbActuator.GetState()
        , Message := 'Not in closed state'
    );

    {analysis -9}
    TEST_FINISHED();
END_IF
END_METHOD

METHOD PRIVATE CloseOneSensorActuatorExpectItToBeClosedWithoutFeedbackVariant2
VAR_INST
    fbActuator : FB_DualPositionActuator
    (
        tActivateTimeout                     := T#5MS
        , tDisableTimeout                    := T#5MS
        , bIsActiveFeedbackSensorAvailable   := TRUE
        , bIsDisabledFeedbackSensorAvailable := FALSE
        , bNormallyDisabled                  := TRUE
    );

    fbTestTimer : TON := (PT := T#2MS);
    bRunOnce    : BOOL;

    nState : INT;
END_VAR
TEST('CloseOneSensorActuatorExpectItToBeClosedWithoutFeedbackVariant2');
fbTestTimer(IN := TRUE);

IF NOT bRunOnce THEN
    bRunOnce := TRUE;
    fbActuator.Disable();
END_IF

CASE nState OF
    0:
        fbActuator(bActiveFeedback := TRUE, bDisableFeedback := FALSE);
        nState := nState + 1;

    1:
        fbActuator(bActiveFeedback := FALSE, bDisableFeedback := FALSE);
END_CASE

IF fbTestTimer.Q THEN
    AssertEquals_INT
    (
        Expected  := E_DualPositionActuatorState.Disabled
        , Actual  := fbActuator.GetState()
        , Message := 'Not in closed state'
    );

    {analysis -9}
    TEST_FINISHED();
END_IF
END_METHOD

METHOD PRIVATE CloseOneSensorActuatorExpectItToTimeout
VAR_INST
    fbActuator : FB_DualPositionActuator
    (
        tActivateTimeout                     := T#10MS
        , tDisableTimeout                    := T#10MS
        , bIsActiveFeedbackSensorAvailable   := FALSE
        , bIsDisabledFeedbackSensorAvailable := TRUE
        , bNormallyDisabled                  := TRUE
    );
    bRunOnce    : BOOL;
    fbTestTimer : TON := (IN := TRUE, PT := T#20MS);
END_VAR
TEST('CloseOneSensorActuatorExpectItToTimeout');

IF NOT bRunOnce THEN
    fbActuator.Disable();
    bRunOnce := TRUE;
    AssertEquals_INT
    (
        Expected  := E_DualPositionActuatorState.Disabling
        , Actual  := fbActuator.GetState()
        , Message := 'Should be closing'
    );
END_IF

fbActuator(bActiveFeedback := FALSE, bDisableFeedback := FALSE);

fbTestTimer();

IF fbTestTimer.Q THEN
    AssertEquals_INT
    (
        Expected  := E_DualPositionActuatorState.TimeoutDisabling
        , Actual  := fbActuator.GetState()
        , Message := 'Should be timeout closing'
    );

    {analysis -9}
    TEST_FINISHED();
END_IF
END_METHOD

METHOD PRIVATE CloseTwoSensorActuatorExpectCloseOutputToBeTrue
VAR_INST
    fbActuator : FB_DualPositionActuator
    (
        tActivateTimeout                     := T#10MS
        , tDisableTimeout                    := T#10MS
        , bIsActiveFeedbackSensorAvailable   := TRUE
        , bIsDisabledFeedbackSensorAvailable := TRUE
        , bNormallyDisabled                  := TRUE
    );
    bRunOnce : BOOL;
END_VAR
TEST('CloseTwoSensorActuatorExpectCloseOutputToBeTrue');

IF NOT bRunOnce THEN
    fbActuator.Disable();
    bRunOnce := TRUE;
END_IF

fbActuator(bActiveFeedback := FALSE, bDisableFeedback := FALSE);

AssertFalse(Condition := fbActuator.bActivate, Message := 'Output is not false');
AssertTrue(Condition := fbActuator.bDisable, Message := 'Output is not true');

{analysis -9}
TEST_FINISHED();
END_METHOD

METHOD PRIVATE CloseTwoSensorActuatorExpectItToBeClosed
VAR_INST
    fbActuator : FB_DualPositionActuator
    (
        tActivateTimeout                     := T#10MS
        , tDisableTimeout                    := T#10MS
        , bIsActiveFeedbackSensorAvailable   := TRUE
        , bIsDisabledFeedbackSensorAvailable := TRUE
        , bNormallyDisabled                  := TRUE
    );
    bRunOnce : BOOL;
END_VAR
TEST('CloseTwoSensorActuatorExpectItToBeClosed');

IF NOT bRunOnce THEN
    fbActuator.Disable();
    bRunOnce := TRUE;
END_IF

fbActuator(bActiveFeedback := FALSE, bDisableFeedback := TRUE);

AssertEquals_INT
(
    Expected  := E_DualPositionActuatorState.Disabled
    , Actual  := fbActuator.GetState()
    , Message := 'Is not closed'
);

{analysis -9}
TEST_FINISHED();
END_METHOD

METHOD PRIVATE CloseTwoSensorActuatorExpectItToTimeout
VAR_INST
    fbActuator : FB_DualPositionActuator
    (
        tActivateTimeout                     := T#5MS
        , tDisableTimeout                    := T#5MS
        , bIsActiveFeedbackSensorAvailable   := TRUE
        , bIsDisabledFeedbackSensorAvailable := TRUE
        , bNormallyDisabled                  := TRUE
    );
    bRunOnce    : BOOL;
    fbTestTimer : TON := (IN := TRUE, PT := T#20MS);
END_VAR
TEST('CloseTwoSensorActuatorExpectItToTimeout');

IF NOT bRunOnce THEN
    fbActuator.Disable();
    bRunOnce := TRUE;
    AssertEquals_INT
    (
        Expected  := E_DualPositionActuatorState.Disabling
        , Actual  := fbActuator.GetState()
        , Message := 'Should be closing'
    );
END_IF

fbActuator(bActiveFeedback := FALSE, bDisableFeedback := FALSE);

fbTestTimer();

IF fbTestTimer.Q THEN
    AssertEquals_INT
    (
        Expected  := E_DualPositionActuatorState.TimeoutDisabling
        , Actual  := fbActuator.GetState()
        , Message := 'Should be timeout closing'
    );

    {analysis -9}
    TEST_FINISHED();
END_IF
END_METHOD

METHOD PRIVATE DisableFeedbackSensorAvailableButNotActiveFeedbackAvailableIfNoDisableFeedbackProvidedItShouldGoToActive
VAR_INST
    fbActuator : FB_DualPositionActuator
    (
        tActivateTimeout                     := T#5MS
        , tDisableTimeout                    := T#5MS
        , bIsActiveFeedbackSensorAvailable   := FALSE
        , bIsDisabledFeedbackSensorAvailable := TRUE
        , bNormallyDisabled                  := TRUE
    );
    nTestState : INT;
END_VAR
TEST('DisableFeedbackSensorAvailableButNotActiveFeedbackAvailableIfNoDisableFeedbackProvidedItShouldGoToActive');

CASE nTestState OF
    0:
        fbActuator(bDisableFeedback := TRUE);
        AssertEquals_INT
        (
            Expected  := E_DualPositionActuatorState.Disabled
            , Actual  := fbActuator.GetState()
            , Message := 'Actuator should be disabled'
        );

        nTestState := nTestState + 1;

    1:
        fbActuator(bDisableFeedback := FALSE);
        AssertEquals_INT
        (
            Expected  := E_DualPositionActuatorState.Active
            , Actual  := fbActuator.GetState()
            , Message := 'Actuator should be active'
        );

        nTestState := nTestState + 1;
    2:
        {analysis -9}
        TEST_FINISHED();
END_CASE
END_METHOD

METHOD PRIVATE DisableTwoSensorNormallyEnabledActuatorExpectItToTimeoutThenExpectDisablingToGoLow
VAR_INST
    fbActuator : FB_DualPositionActuator
    (
        tActivateTimeout                     := T#10MS
        , tDisableTimeout                    := T#10MS
        , bIsActiveFeedbackSensorAvailable   := TRUE
        , bIsDisabledFeedbackSensorAvailable := TRUE
        , bNormallyDisabled                  := FALSE
    );
    bRunOnce    : BOOL;
    fbTestTimer : TON := (IN := TRUE, PT := T#20MS);
    nTestStep   : INT;
END_VAR
TEST('DisableTwoSensorNormallyEnabledActuatorExpectItToTimeoutThenExpectDisablingToGoLow');
fbActuator(bActiveFeedback := FALSE, bDisableFeedback := FALSE);
fbTestTimer();

IF NOT bRunOnce THEN
    fbActuator.Disable();
    bRunOnce := TRUE;
END_IF

CASE nTestStep OF
    0:
        IF fbTestTimer.ET = T#5MS THEN
            nTestStep := nTestStep + 1;
        END_IF

    1:
        AssertEquals_INT
        (
            Expected  := E_DualPositionActuatorState.Disabling
            , Actual  := fbActuator.GetState()
            , Message := 'Should be disabling'
        );

        AssertTrue(fbActuator.bDisable, Message := 'Actuator should disable');
        nTestStep := nTestStep + 1;

    2:
// Do nothing
END_CASE

IF fbTestTimer.Q THEN
    AssertEquals_INT(Expected := 2, Actual := nTestStep, Message := 'Not correct step');
    AssertEquals_INT
    (
        Expected  := E_DualPositionActuatorState.TimeoutDisabling
        , Actual  := fbActuator.GetState()
        , Message := 'Should be timeout disabling'
    );

    AssertFalse(fbActuator.bDisable, Message := 'Actuator should not disable');
    {analysis -9}
    TEST_FINISHED();
END_IF
END_METHOD

METHOD PRIVATE EnableTwoSensorNormallyDisabledActuatorExpectItToTimeoutThenExpectActuationToGoLow
VAR_INST
    fbActuator : FB_DualPositionActuator
    (
        tActivateTimeout                     := T#10MS
        , tDisableTimeout                    := T#10MS
        , bIsActiveFeedbackSensorAvailable   := TRUE
        , bIsDisabledFeedbackSensorAvailable := TRUE
        , bNormallyDisabled                  := TRUE
    );
    bRunOnce    : BOOL;
    fbTestTimer : TON := (IN := TRUE, PT := T#20MS);
    nTestStep   : INT;
END_VAR
TEST('EnableTwoSensorNormallyDisabledActuatorExpectItToTimeoutThenExpectActuationToGoLow');
fbActuator(bActiveFeedback := FALSE, bDisableFeedback := FALSE);
fbTestTimer();

IF NOT bRunOnce THEN
    fbActuator.Activate();
    bRunOnce := TRUE;
END_IF

CASE nTestStep OF
    0:
        IF fbTestTimer.ET = T#5MS THEN
            nTestStep := nTestStep + 1;
        END_IF

    1:
        AssertEquals_INT
        (
            Expected  := E_DualPositionActuatorState.Activating
            , Actual  := fbActuator.GetState()
            , Message := 'Should be enabling'
        );

        AssertTrue(fbActuator.bActivate, Message := 'Actuator should actuate');
        nTestStep := nTestStep + 1;

    2:
// Do nothing
END_CASE

IF fbTestTimer.Q THEN
    AssertEquals_INT(Expected := 2, Actual := nTestStep, Message := 'Not correct step');
    AssertEquals_INT
    (
        Expected  := E_DualPositionActuatorState.TimeoutActivating
        , Actual  := fbActuator.GetState()
        , Message := 'Should be timeout activating'
    );

    AssertFalse(fbActuator.bActivate, Message := 'Actuator should not actuate');
    {analysis -9}
    TEST_FINISHED();
END_IF
END_METHOD

METHOD PRIVATE GivenActivatedFeedBackSensorNotAvailableAndNormallyActivatedThenShouldBeActivated
VAR
    fbDualPositionActuator : FB_DualPositionActuator
    (
        tActivateTimeout                     := T#0S
        , tDisableTimeout                    := T#0S
        , bIsActiveFeedbackSensorAvailable   := FALSE
        , bIsDisabledFeedbackSensorAvailable := TRUE
        , bNormallyDisabled                  := FALSE
    );
END_VAR
TEST('GivenActivatedFeedBackSensorNotAvailableAndNormallyActivatedThenShouldBeActivated');

fbDualPositionActuator(bActiveFeedback := FALSE, bDisableFeedback := FALSE);

AssertEquals_INT
(
    Expected  := E_DualPositionActuatorState.Active
    , Actual  := fbDualPositionActuator.GetState()
    , Message := 'Not in active state'
);

{analysis -9}
TEST_FINISHED();
END_METHOD

METHOD PRIVATE GivenDisabledFeedBackSensorNotAvailableAndNormallyDisabledThenShouldBeDisabled
VAR
    fbDualPositionActuator : FB_DualPositionActuator
    (
        tActivateTimeout                     := T#0S
        , tDisableTimeout                    := T#0S
        , bIsActiveFeedbackSensorAvailable   := TRUE
        , bIsDisabledFeedbackSensorAvailable := FALSE
        , bNormallyDisabled                  := TRUE
    );
END_VAR
TEST('GivenDisabledFeedBackSensorNotAvailableAndNormallyDisabledThenShouldBeDisabled');

fbDualPositionActuator(bActiveFeedback := FALSE, bDisableFeedback := FALSE);

AssertEquals_INT
(
    Expected  := E_DualPositionActuatorState.Disabled
    , Actual  := fbDualPositionActuator.GetState()
    , Message := 'Not in disabled state'
);

{analysis -9}
TEST_FINISHED();
END_METHOD

METHOD PRIVATE OpenOneSensorActuatorExpectItToBeOpenWithoutFeedback
VAR_INST
    fbActuator : FB_DualPositionActuator
    (
        tActivateTimeout                     := T#5MS
        , tDisableTimeout                    := T#5MS
        , bIsActiveFeedbackSensorAvailable   := FALSE
        , bIsDisabledFeedbackSensorAvailable := TRUE
        , bNormallyDisabled                  := TRUE
    );

    fbTestTimer : TON := (PT := T#2MS);
    bRunOnce    : BOOL;
END_VAR
TEST('OpenOneSensorActuatorExpectItToBeOpenWithoutFeedback');
fbTestTimer(IN := TRUE);

IF NOT bRunOnce THEN
    bRunOnce := TRUE;
    fbActuator.Activate();
END_IF

fbActuator(bActiveFeedback := FALSE, bDisableFeedback := FALSE);

IF fbTestTimer.Q THEN
    AssertEquals_INT
    (
        Expected  := E_DualPositionActuatorState.Active
        , Actual  := fbActuator.GetState()
        , Message := 'Not in open state'
    );

    {analysis -9}
    TEST_FINISHED();
END_IF
END_METHOD

METHOD PRIVATE OpenOneSensorActuatorExpectItToBeOpenWithoutFeedbackVariant2
VAR_INST
    fbActuator : FB_DualPositionActuator
    (
        tActivateTimeout                     := T#5MS
        , tDisableTimeout                    := T#5MS
        , bIsActiveFeedbackSensorAvailable   := FALSE
        , bIsDisabledFeedbackSensorAvailable := TRUE
        , bNormallyDisabled                  := TRUE
    );

    fbTestTimer : TON := (PT := T#2MS);
    bRunOnce    : BOOL;

    nState : INT;
END_VAR
TEST('OpenOneSensorActuatorExpectItToBeOpenWithoutFeedbackVariant2');
fbTestTimer(IN := TRUE);

IF NOT bRunOnce THEN
    bRunOnce := TRUE;
    fbActuator.Activate();
END_IF

CASE nState OF
    0:
        fbActuator(bActiveFeedback := FALSE, bDisableFeedback := TRUE);
        nState := nState + 1;

    1:
        fbActuator(bActiveFeedback := FALSE, bDisableFeedback := FALSE);
END_CASE

IF fbTestTimer.Q THEN
    AssertEquals_INT
    (
        Expected  := E_DualPositionActuatorState.Active
        , Actual  := fbActuator.GetState()
        , Message := 'Not in open state'
    );

    {analysis -9}
    TEST_FINISHED();
END_IF
END_METHOD

METHOD PRIVATE OpenOneSensorActuatorExpectItToTimeout
VAR_INST
    fbActuator : FB_DualPositionActuator
    (
        tActivateTimeout                     := T#5MS
        , tDisableTimeout                    := T#5MS
        , bIsActiveFeedbackSensorAvailable   := TRUE
        , bIsDisabledFeedbackSensorAvailable := FALSE
        , bNormallyDisabled                  := TRUE
    );
    bRunOnce    : BOOL;
    fbTestTimer : TON := (IN := TRUE, PT := T#100MS);
END_VAR
TEST('OpenOneSensorActuatorExpectItToTimeout');
fbActuator(bActiveFeedback := FALSE, bDisableFeedback := FALSE);

IF NOT bRunOnce THEN
    fbActuator.Activate();
    bRunOnce := TRUE;
    AssertEquals_INT
    (
        Expected  := E_DualPositionActuatorState.Activating
        , Actual  := fbActuator.GetState()
        , Message := 'Should be opening'
    );
END_IF

IF fbTestTimer.ET = T#3MS THEN
    AssertEquals_INT
    (
        Expected  := E_DualPositionActuatorState.Activating
        , Actual  := fbActuator.GetState()
        , Message := 'Should be opening'
    );
END_IF

fbTestTimer();

IF fbTestTimer.Q THEN
    AssertEquals_INT
    (
        Expected  := E_DualPositionActuatorState.TimeoutActivating
        , Actual  := fbActuator.GetState()
        , Message := 'Should be timeout extended'
    );

    {analysis -9}
    TEST_FINISHED();
END_IF
END_METHOD

METHOD PRIVATE OpenTwoSensorActuatorExpectItToBeOpen
VAR_INST
    fbActuator : FB_DualPositionActuator
    (
        tActivateTimeout                     := T#10MS
        , tDisableTimeout                    := T#10MS
        , bIsActiveFeedbackSensorAvailable   := TRUE
        , bIsDisabledFeedbackSensorAvailable := TRUE
        , bNormallyDisabled                  := TRUE
    );
    nState : INT;
END_VAR
TEST('OpenTwoSensorActuatorExpectItToBeOpen');

CASE nState OF
    0:
        fbActuator.Activate();
        nState := 10;

    10:
        fbActuator.bActiveFeedback  := FALSE;
        fbActuator.bDisableFeedback := FALSE;
        nState                      := 20;

    20:
        AssertEquals_INT
        (
            Expected  := E_DualPositionActuatorState.Activating
            , Actual  := fbActuator.GetState()
            , Message := 'Is not opening'
        );

        nState := 30;

    30:
        fbActuator.bActiveFeedback  := TRUE;
        fbActuator.bDisableFeedback := FALSE;
        nState                      := 40;

    40:
        AssertEquals_INT
        (
            Expected  := E_DualPositionActuatorState.Active
            , Actual  := fbActuator.GetState()
            , Message := 'Is not open'
        );

        {analysis -9}
        TEST_FINISHED();
END_CASE

fbActuator();
END_METHOD

METHOD PRIVATE OpenTwoSensorActuatorExpectItToTimeout
VAR_INST
    fbActuator : FB_DualPositionActuator
    (
        tActivateTimeout                     := T#5MS
        , tDisableTimeout                    := T#5MS
        , bIsActiveFeedbackSensorAvailable   := TRUE
        , bIsDisabledFeedbackSensorAvailable := TRUE
        , bNormallyDisabled                  := TRUE
    );
    bRunOnce    : BOOL;
    fbTestTimer : TON := (IN := TRUE, PT := T#15MS);
END_VAR
TEST('OpenTwoSensorActuatorExpectItToTimeout');
fbActuator(bActiveFeedback := FALSE, bDisableFeedback := FALSE);

IF NOT bRunOnce THEN
    fbActuator.Activate();
    bRunOnce := TRUE;
    AssertEquals_INT
    (
        Expected  := E_DualPositionActuatorState.Activating
        , Actual  := fbActuator.GetState()
        , Message := 'Should be opening'
    );
END_IF

IF fbTestTimer.ET = T#3MS THEN
    AssertEquals_INT
    (
        Expected  := E_DualPositionActuatorState.Activating
        , Actual  := fbActuator.GetState()
        , Message := 'Should be opening'
    );
END_IF

fbTestTimer();

IF fbTestTimer.Q THEN
    AssertEquals_INT
    (
        Expected  := E_DualPositionActuatorState.TimeoutActivating
        , Actual  := fbActuator.GetState()
        , Message := 'Should be timeout extended'
    );

    {analysis -9}
    TEST_FINISHED();
END_IF
END_METHOD

END_FUNCTION_BLOCK

// ---- Test/Ats400_Etl_Tests/InputAts400_Test.TcPOU
FUNCTION_BLOCK InputAts400_Test EXTENDS TcUnit.FB_TestSuite
VAR

END_VAR

ParseVariantOne();

METHOD PRIVATE ParseVariantOne
VAR
    aInput : ARRAY[1..8] OF BOOL;

    input : InputAts400;

    inputData : InputDataAts400;
    i         : UINT;
END_VAR
VAR CONSTANT
    lower : UINT := 1;
    upper : UINT := 8;
END_VAR
Test('ParseVariantOne');

input(input := aInput);
// just for validation an example
AssertFalse(Condition := inputData.ContactExits, 'Contact Exits muss falsch sein');

FOR i := lower TO upper DO
    aInput[i] := TRUE;
END_FOR

input(input := aInput);

inputData := input.GetInputData();
AssertTrue(Condition := inputData.Pass, ' Pass must be true');
AssertTrue(Condition := inputData.Fail, ' Fail must be true');
AssertTrue(Condition := inputData.InOp, ' In Op must be true');
AssertTrue(Condition := inputData.ResultImpuls, ' Result Impuls must be true');
AssertTrue(Condition := inputData.DummyOut, 'Dummy Out must be true');
AssertTrue(Condition := inputData.Ready, 'Ready must be true');
AssertTrue(Condition := inputData.SafetyCircuit, 'Safety must be true');
AssertTrue(Condition := inputData.ContactExits, 'KontaktExists must be true');

TEST_FINISHED();
END_METHOD

END_FUNCTION_BLOCK

// ---- POUs/ATS400_ETL/FunctionBlocks/InputAts400.TcPOU
FUNCTION_BLOCK InputAts400 IMPLEMENTS IInputAts400
VAR_INPUT
    input : ARRAY[1..8] OF BOOL;
END_VAR

METHOD GetInputData : InputDataAts400
VAR_INPUT
END_VAR
GetInputData.Pass          := input[1];
GetInputData.Fail          := input[2];
GetInputData.InOp          := input[3];
GetInputData.ResultImpuls  := input[4];
GetInputData.DummyOut      := input[5];
GetInputData.Ready         := input[6];
GetInputData.SafetyCircuit := input[7];
GetInputData.ContactExits  := input[8];
END_METHOD

END_FUNCTION_BLOCK

// ---- Test/Ats400_Etl_Tests/OutputAts400_Test.TcPOU
FUNCTION_BLOCK OutputAts400_Test EXTENDS FB_TestSuite IMPLEMENTS TcoCore.ITcoContext
VAR
    //Context for TcOpen
    _nfContext : TcoCore.TcoContextNfCompatibility;

    timer : ton := (pt := T#15MS); //mind 18ms muss Select gesetzt sein
END_VAR
VAR
    dut : OutputAts400(THIS^, eRestoreMode.None);
END_VAR

VAR
    dut_Select : OutputAts400(THIS^, eRestoreMode.None);

    input          : InputAts400MockStatusReady;
    itfInputAts400 : IInputAts400 := input;
    inData         : InputDataAts400;
END_VAR

VAR
    dut_bitCombi  : OutputAts400(THIS^, eRestoreMode.None);
    timerBitCombi : TON := (PT := T#15MS);
END_VAR

VAR
    dut_bitCombi9  : OutputAts400(THIS^, eRestoreMode.None);
    timerBitCombi9 : TON := (PT := T#15MS);
END_VAR

_nfContext.VolatileOpen(); //Required for TCopen
////==============================================

SetOutputsAndVerify();
SetProgram5_ExpectBit1TrueBit2FalseBit3TrueOthersFalse();
SetDifferentPrograms_ExpectCorrespondingBitCombination();
SetDifferentProgramsLike9_ExpectCorrespondingBitCombination();
////==============================================
_nfContext.VolatileClose();

PROPERTY Context : TcoCore.ITcoContext
GET
Context := This^._nfContext;
END_GET
END_PROPERTY

PROPERTY EndCycleCount : ULINT
GET
EndCycleCount := THIS^._nfContext._endCycleCount;
END_GET
END_PROPERTY

PROPERTY Environment : TcoCore.ITcoContextEnvironment
GET
Environment := THIS^._nfContext._settings;
END_GET
END_PROPERTY

PROPERTY Identity : ULINT
GET
Identity := THIS^._nfContext._Identity;
END_GET
END_PROPERTY

PROPERTY Logger : TcoCore.ITcoLogger
GET
Logger := THIS^._nfContext._logger;
END_GET
END_PROPERTY

PROPERTY RealTimeClock : TcoCore.ITcoRtc
GET
RealTimeClock := THIS^._nfContext._rtc;
END_GET
END_PROPERTY

METHOD PRIVATE SetDifferentPrograms_ExpectCorrespondingBitCombination
VAR_INST
    selectedProgram : UINT := 11;
END_VAR
TEST('SetDifferentPrograms_ExpectCorrespondingBitCombination');

timerBitCombi(in := TRUE);

dut_bitCombi.SelectProgramm(selectedProgram);

IF timerBitCombi.Q THEN
    timer(in := false);
    AssertTrue(Condition := dut_bitCombi.output[6], 'Select must be true');
    AssertTrue(Condition := dut_bitCombi.output[7], 'Bit1 must be true');
    AssertTrue(Condition := dut_bitCombi.output[8], 'Bit2 must be true');
    AssertFalse(Condition := dut_bitCombi.output[9], 'Bit3 must be true');
    AssertTrue(Condition := dut_bitCombi.output[10], 'Bit4 must be true');
    AssertFalse(Condition := dut_bitCombi.output[11], 'Bit5 must be false');
    AssertFalse(Condition := dut_bitCombi.output[12], 'Bit6 must be false');

END_IF

IF dut_bitCombi.SelectProgramm(programm := selectedProgram).Done THEN
    TEST_FINISHED();
END_IF
END_METHOD

METHOD PRIVATE SetDifferentProgramsLike9_ExpectCorrespondingBitCombination
VAR_INST
    selectedProgram : UINT := 9;
END_VAR
TEST('SetDifferentProgramsLike9_ExpectCorrespondingBitCombination');

timerBitCombi9(in := TRUE);

dut_bitCombi9.SelectProgramm(selectedProgram);

IF timerBitCombi9.Q THEN
    timer(in := false);
    AssertTrue(Condition := dut_bitCombi9.output[6], 'Select must be true');
    AssertTrue(Condition := dut_bitCombi9.output[7], 'Bit1 must be true');
    AssertFalse(Condition := dut_bitCombi9.output[8], 'Bit2 must be false');
    AssertFalse(Condition := dut_bitCombi9.output[9], 'Bit3 must be false');
    AssertTrue(Condition := dut_bitCombi9.output[10], 'Bit4 must be true');
    AssertFalse(Condition := dut_bitCombi9.output[11], 'Bit5 must be false');
    AssertFalse(Condition := dut_bitCombi9.output[12], 'Bit6 must be false');

END_IF

IF dut_bitCombi9.SelectProgramm(programm := selectedProgram).Done THEN
    TEST_FINISHED();
END_IF
END_METHOD

METHOD PRIVATE SetOutputsAndVerify
TEST('SetOutputsAndVerify');

dut.Start(TRUE);
AssertTrue(Condition := dut.output[1], 'Start shall be true');
dut.Start(FALSE);

dut.AbortTest(TRUE);
AssertTrue(Condition := dut.output[2], 'Abort shall be true');
dut.AbortTest(FALSE);

dut.SetManualPass(TRUE);
AssertTrue(Condition := dut.output[3], 'SetManualPass shall be true');
dut.SetManualPass(FALSE);

dut.SetManualFail(TRUE);
AssertTrue(Condition := dut.output[4], 'SetManualFail shall be true');
dut.SetManualFail(FALSE);

dut.SetDummyReady(TRUE);
AssertTrue(Condition := dut.output[5], 'SetDummyReady shall be true');
dut.SetDummyReady(FALSE);

timer(in := TRUE);
dut.SelectProgramm(3);
//AssertTrue(Condition := out.out[6], 'Select must be true');
//AssertFalse(Condition := out.out[7], 'Bits muessen false sein');

IF timer.Q THEN
    AssertTrue(Condition := dut.output[6], 'Select must be true');

    AssertTrue(Condition := dut.output[7], 'Bit1 must be true');
    AssertTrue(Condition := dut.output[8], 'Bit2 must be true');
    AssertFalse(Condition := dut.output[9], 'Bit3 must be false');
    AssertFalse(Condition := dut.output[10], 'Bit4 must be false');
    AssertFalse(Condition := dut.output[11], 'Bit5 must be false');
    AssertFalse(Condition := dut.output[12], 'Bit6 must be false');

    TEST_FINISHED();
END_IF
END_METHOD

METHOD PRIVATE SetProgram5_ExpectBit1TrueBit2FalseBit3TrueOthersFalse
VAR_INST
    duration        : TON  := (pt := T#50MS);
    selectedProgram : UINT := 5;
END_VAR
TEST('SetProgram5_ExpectBit1TrueBit2FalseBit3TrueOthersFalse');

// Offen, weis nicht, wie das funktioniert
//Out 3
//Ausgang IN OP
//Digitale Ausgabe zur Rückmeldung einer aktiven sicherheitstechnischen Prüfung des Prüfsystems.
// Zwischen den einzelnen Prüfungen wechselt das Bit von 1 auf 0.

duration(in := TRUE);

inData := itfInputAts400.GetInputData();
AssertTrue(inData.Ready, 'Ready muss true sein, sonst kann kein Programm gewechselt werden');

dut_Select.SelectProgramm(selectedProgram);

IF duration.ET >= T#4MS AND duration.ET <= T#30MS THEN
    AssertTrue(Condition := dut.output[6], 'Start, Select must be true ');

    AssertTrue(Condition := dut_Select.output[7], 'Start,Bit1 must be true');
    AssertFalse(Condition := dut_Select.output[8], 'Start,Bit2 must be false');
    AssertTrue(Condition := dut_Select.output[9], 'Start,Bit3 must be true');
    AssertFalse(Condition := dut_Select.output[10], 'Start,Bit4 must be false');
    AssertFalse(Condition := dut_Select.output[11], 'Start,Bit5 must be false');
    AssertFalse(Condition := dut_Select.output[12], 'Start,Bit6 must be false');

end_if

IF duration.ET >= T#22MS AND duration.ET <= T#30MS THEN
    // muss immer noch true sein
    AssertTrue(Condition := dut_Select.output[6], 'Still, Select must be true');

    AssertTrue(Condition := dut_Select.output[7], 'Still,Bit1 must be true');
    AssertFalse(Condition := dut_Select.output[8], 'Still,Bit2 must be false');
    AssertTrue(Condition := dut_Select.output[9], 'Still,Bit3 must be true');
    AssertFalse(Condition := dut_Select.output[10], 'Still,Bit4 must be false');
    AssertFalse(Condition := dut_Select.output[11], 'Still,Bit5 must be false');
    AssertFalse(Condition := dut_Select.output[12], 'Still,Bit6 must be false');

END_IF

IF dut_Select.SelectProgramm(programm := selectedProgram).Done THEN
    AssertFalse(Condition := dut_Select.output[6], 'Alles False');

    AssertFalse(Condition := dut_Select.output[7], 'Alles False');
    AssertFalse(Condition := dut_Select.output[8], 'Alles False');
    AssertFalse(Condition := dut_Select.output[9], 'Alles False');
    AssertFalse(Condition := dut_Select.output[10], 'Alles False');
    AssertFalse(Condition := dut_Select.output[11], 'Alles False');
    AssertFalse(Condition := dut_Select.output[12], 'Alles False');

    TEST_FINISHED();
END_IF
END_METHOD

PROPERTY StartCycleCount : ULINT
GET
StartCycleCount := THIS^._nfContext._startCycleCount;
END_GET
END_PROPERTY

END_FUNCTION_BLOCK

// ---- POUs/ATS400_ETL/FunctionBlocks/OutputAts400.TcPOU
FUNCTION_BLOCK OutputAts400 EXTENDS TcoCore.TcoState IMPLEMENTS IOutputAts400
VAR_OUTPUT
    output : ARRAY[1..12] OF BOOl;
END_VAR
VAR
    selectProgramTask : SelectProgramTask(THIS^);
END_VAR

METHOD AbortTest
VAR_INPUT
    enable : BOOL;
END_VAR
THIS^.output[2] := enable;
END_METHOD

METHOD SelectProgramm : TcoCore.ITcoTaskStatus
VAR_INPUT
    programm : UINT;
END_VAR
//mind 18ms muss Select gesetzt sein

SelectProgramm := selectProgramTask.Invoke();
selectProgramTask(selectedProgram := programm, output => output);
END_METHOD

METHOD SetDummyReady
VAR_INPUT
    enable : BOOL;
END_VAR
output[5] := enable;
END_METHOD

METHOD SetManualFail
VAR_INPUT
    enable : BOOL;
END_VAR
output[4] := enable;
END_METHOD

METHOD SetManualPass
VAR_INPUT
    enable : BOOL;
END_VAR
output[3] := enable;
END_METHOD

METHOD Start
VAR_INPUT
    enable : BOOL;
END_VAR
this^.output[1] := enable;
END_METHOD

END_FUNCTION_BLOCK

// ---- POUs/ATS400_ETL/FunctionBlocks/SelectProgramTask.TcPOU
FUNCTION_BLOCK SelectProgramTask EXTENDS TcoCore.TcoTask
VAR_OUTPUT
    {attribute clr [RenderIgnore()]}
    output : ARRAY[lower..upper] OF BOOL;
END_VAR

VAR_INPUT
    {attribute addProperty Name "<#Waehle ein Programm#>"}
    selectedProgram : UINT;
END_VAR

VAR
    {attribute clr [RenderIgnore()]}
    i : UINT;
    //~
    selectState : (Init
        , Abort
        , Select
        , SetOutput
        , Reset);
    //~
    //~
    timer : TON := (PT := T#18MS); //18ms mind. for Select Active
    //~
END_VAR

VAR CONSTANT
    {attribute clr [RenderIgnore()]}
    lower : UINT := 1;
    {attribute clr [RenderIgnore()]}
    upper : UINT := 12;
END_VAR

IF (THIS^.Execute()) THEN
    timer();

    CASE selectState OF
        Init:
            selectState := Abort;
        Abort:
            output[2] := TRUE;
            timer(In := TRUE, pt := T#1MS);

            IF timer.Q THEN
                output[2]   := FALSE;
                selectState := Select;
                timer(In := FALSE);
            END_IF
        Select:
            timer(In := TRUE, PT := T#50MS);
            output[6]   := TRUE;
            selectState := SetOutput;
        SetOutPut:
            output[7]  := (selectedProgram.0);
            output[8]  := (selectedProgram.1);
            output[9]  := (selectedProgram.2);
            output[10] := (selectedProgram.3);
            output[11] := (selectedProgram.4);
            output[12] := (selectedProgram.5);

            IF timer.Q THEN
                selectState := Reset;
            end_if
        Reset:
            output[6]  := FALSE;
            output[7]  := FALSE;
            output[8]  := FALSE;
            output[9]  := FALSE;
            output[10] := FALSE;
            output[11] := FALSE;
            output[12] := FALSE;

            timer(In := FALSE);
            THIS^.DoneWhen(TRUE);
    END_CASE

END_IF

(*~
    <docu>
        <summary>
            Executes ones when the task starts (at the moment of transition from the ```Requested``` state into the ```Busy``` state).
        </summary>
    </docu>
~*)
METHOD PROTECTED OnStart
timer(in := FALSE);
END_METHOD

END_FUNCTION_BLOCK

// ---- POUs/ATS400_ETL/Mocks/InputAts400MockStatusReady.TcPOU
FUNCTION_BLOCK InputAts400MockStatusReady IMPLEMENTS IInputAts400

METHOD GetInputData : InputDataAts400
GetInputData.Ready := true;
END_METHOD

END_FUNCTION_BLOCK

// ---- POUs/Communication Extern/FunctionBlocks/CommunicationRoboterOmron.TcPOU
FUNCTION_BLOCK CommunicationRoboterOmron IMPLEMENTS ICommunicationRoboterOmron
VAR
    comRobseq     : TcpIpCommSeq(sRemoteHost := _sRemoteHost, serverPort := _serverPort);
    itfCommRobSeq : ICommSeq := comRobseq;
    msgToSend     : uTelegrammOmronTcp;
    msgReceive    : uTelegrammOmronTcp;

    _sRemoteHost : STRING;
    _serverPort  : UDINT;

    _msgFmtStr : T_MaxString;
    _eState    : E_SocketConnectionState := eSOCKET_DISCONNECTED;
END_VAR
VAR
    inCom : InCommunicationRobOmron;
END_VAR
VAR
    outCom : OutCommunicationRobOmron;
END_VAR

METHOD ContactPrepared
VAR_INPUT
    enable : BOOL;
END_VAR
outCom.ContactPrepared := enable;
END_METHOD

{warning 'add property implementation'}
PROPERTY EState : Tc2_TcpIp.E_SocketConnectionState
GET
Estate := _eState;
END_GET
END_PROPERTY

METHOD FB_init : BOOL
VAR_INPUT
    bInitRetains : BOOL; // if TRUE, the retain variables are initialized (warm start / cold start)
    bInCopyCode : BOOL;  // if TRUE, the instance afterwards gets moved into the copy code (online change)
    sRemoteHost : STRING;
    serverPort : UDINT;
END_VAR
_sRemoteHost := sRemoteHost;
_serverPort  := serverPort;
comRobseq.FB_init
(
    bInitRetains  := bInitretains
    , bInCopyCode := bInCopyCode
    , sRemoteHost := sRemoteHost
    , serverPort  := serverPort
);
END_METHOD

METHOD HighPowerOff
VAR_INPUT
    enable : BOOL;
END_VAR
outCom.HighPowerOff := enable;
END_METHOD

METHOD HighPowerOn
VAR_INPUT
    enable : BOOL;
END_VAR
outCom.HighPowerOn:= enable;
END_METHOD

METHOD PRIVATE MapCom
//TCP IP Komm
////==========in
inCom.homePosReached := INT_TO_BOOL(msgReceive.stTel.myBool[1]);
inCom.statusRunning  := INT_TO_BOOL(msgReceive.stTel.myBool[2]);
inCom.Fault          := INT_TO_BOOL(msgReceive.stTel.myBool[3]);
inCom.PowerOn        := INT_TO_BOOL(msgReceive.stTel.myBool[4]);
inCom.Estop          := INT_TO_BOOL(msgReceive.stTel.myBool[5]);

inCom.FaultID := msgReceive.stTel.myInt[1];

//===================Outputs===========================================
msgToSend.stTel.myInt[1] := BOOL_TO_INT(outCom.StartAutomatic);
msgToSend.stTel.myInt[2] := BOOL_TO_INT(outCom.stopAutomatic);
msgToSend.stTel.myInt[3] := BOOL_TO_INT(outCom.reset);
msgToSend.stTel.myInt[4] := BOOL_TO_INT(outCom.requestHome);
msgToSend.stTel.myInt[5] := BOOL_TO_INT(outCom.highPowerOn);
msgToSend.stTel.myInt[6] := BOOL_TO_INT(outCom.highPowerOff);
END_METHOD

{warning 'add property implementation'}
PROPERTY MsgFmtStr : Tc2_System.T_MaxString
GET
MsgFmtStr := _msgFmtStr;
END_GET
END_PROPERTY

METHOD RequestHome
VAR_INPUT
    enable : BOOL;
END_VAR
outCom.RequestHome := enable;
END_METHOD

METHOD Reset
VAR_INPUT
    enable : BOOL;
END_VAR
outCom.Reset := enable;
END_METHOD

METHOD Run
itfCommRobSeq.Run(msgSend := msgToSend, msgRcv := msgReceive);
MapCom();
END_METHOD

METHOD StartAutomatic
VAR_INPUT
    enable : BOOL;
END_VAR
outCom.StartAutomatic := enable;
END_METHOD

{attribute 'monitoring' := 'variable'}
PROPERTY StatusCom : REFERENCE TO OutCommunicationRobOmron
GET
//For Testing
StatusCom REF= outCom;
END_GET
END_PROPERTY

METHOD StopAutomatic
VAR_INPUT
    enable : BOOL;
END_VAR
outCom.StopAutomatic := enable;
END_METHOD

END_FUNCTION_BLOCK

// ---- POUs/Communication Extern/FunctionBlocks/TcpIpCommSeq.TcPOU
FUNCTION_BLOCK TcpIpCommSeq IMPLEMENTS ICommSeq
VAR
    msgSend : uTelegrammOmronTcp;
    msgRcv  : uTelegrammOmronTcp;
END_VAR
VAR
    _sRemoteHost     : STRING;
    _serverPort      : UDINT;
    eStep            : E_ConnectionStepsTcp := E_ConnectionStepsTcp.eCONNECTION_STATE_IDLE;
    _bEnable         : BOOL                 := TRUE;
    _comTrig         : Tc2_Standard.f_TRIG;
    _comStatus       : BOOL;
    _bConnected      : BOOL;
    _bDisconnect     : BOOL;
    fbServerCon      : Tc2_TcpIp.FB_ClientServerConnection;
    fbSend           : Tc2_TcpIp.FB_SocketSend;
    fbRceive         : Tc2_TcpIp.FB_SocketReceive;
    cbLen            : UDINT;
    bExecute         : BOOL;
    tTimeout         : TIME                    := T#2S;
    _eState          : E_SocketConnectionState := eSOCKET_DISCONNECTED;
    sSrvNetId        : T_AmsNetId              := '';
    hSocket          : T_HSOCKET;
    bExecuteRec      : BOOL;
    bBusy            : BOOL;
    bError           : BOOL;
    nErrId           : UDINT;
    nRecBytes        : UDINT;
    _hbOld           : INT := 0;
    _hb              : INT;
    _hbErrCoun       : INT;
    index            : uINT;
    _reset           : BOOL;
    fbPollTimer      : Tc2_Standard.TON := (PT := TIME#10MS); (* Receive poll timer *)
    fbReconnectTimer : Tc2_Standard.TON := (pt := TIME#1S);
    fbResponseTimer  : Tc2_Standard.TON := (pt := TIME#160MS); (* Response timeout timer *)
    fbTimeOut        : Tc2_Standard.TON := (pt := TIME#2S);    //Time OUt für ANtwort
    reconnectTime    : TIME             := T#1S;
    _index           : INT              := 0;
    _dataRcv         : Tc2_Standard.R_TRIG;
    _bConnectedTrig  : Tc2_Standard.R_TRIG;
    _n               : INT;
    _ErrorCycle      : UDINT;
    faultID          : UINT;
    _msgFmtStr       : T_MaxString;
END_VAR
VAR CONSTANT
    hbError : INT := 5;
END_VAR

{warning 'add property implementation'}
PROPERTY EState : Tc2_TcpIp.E_SocketConnectionState
GET
Estate := _eState;
END_GET
END_PROPERTY

METHOD FB_init : BOOL
VAR_INPUT
    bInitRetains : BOOL; // if TRUE, the retain variables are initialized (warm start / cold start)
    bInCopyCode : BOOL;  // if TRUE, the instance afterwards gets moved into the copy code (online change)
    sRemoteHost : STRING;
    serverPort : UDINT;
END_VAR
_sRemoteHost := sRemoteHost;
_serverPort  := serverPort;
END_METHOD

METHOD PRIVATE mClearData : BOOL
VAR
    _index : UINT;
END_VAR


FOR _index := 1 TO SIZEOF(TcpIpCommSeq.msgRcv) - 1 DO
    msgRcv.aTel[_index] := 0;
END_FOR
END_METHOD

{warning 'add property implementation'}
PROPERTY MsgFmtStr : Tc2_System.T_MaxString
GET
MsgFmtStr := _msgFmtStr;
END_GET
END_PROPERTY

METHOD Run
VAR_INPUT
    msgSend : REFERENCE TO uTelegrammOmronTcp;
    msgRcv  : REFERENCE TO uTelegrammOmronTcp;
END_VAR
msgSend REF= THIS^.msgSend;
msgRcv  REF= THIS^.msgRcv;

IF NOT _bConnected THEN
    mClearData();
END_IF

IF _comTrig.Q THEN
    //    fbReconnectTimer(pt := T#0MS);
    IF _comStatus THEN
        _comStatus := FALSE;
        _bEnable   := FALSE;
    ELSE
        _bEnable   := TRUE;
        _comStatus := true;
    END_IF

    //else
    //    fbReconnectTimer(pt := t#5s);
END_IF

//StateMachine f+ür die TCP/IP Com
//Solange Enable true, versucht der Baustein eine Verbindung aufzubauen
//Gesamte Zeitüberwachung für bEnable und keine Verbindung, -> als Error an HMI
fbPollTimer(in := NOT fbPollTimer.Q);
fbResponseTimer(in := NOT fbResponseTimer.Q);

CASE eStep OF
    eCONNECTION_STATE_IDLE:
        IF _bEnable XOR _bConnected THEN
            IF _bEnable THEN
                fbReconnectTimer(in := TRUE);

                IF fbReconnectTimer.Q THEN
                    _bDisconnect := FALSE;
                    nRecBytes    := 0;
                    fbReconnectTimer(in := FALSE, pt := reconnectTime);
                    estep := eCONNECTION_STATE_CONNECT_START;
                END_IF
            ELSE
                estep := eCONNECTION_STATE_CLOSE_START;
            END_IF
        ELSIF _bConnected THEN
            estep := eCONNECTION_STATE_DATAEXCHANGE;
        ELSE
            fbReconnectTimer(in := FALSE);
        END_IF
    eCONNECTION_STATE_CONNECT_START:
        cbLen := SIZEOF(msgSend.aTel) + 1;
        //Rücksetzten Heartbeat
        _hb        := 0;
        _hbOld     := 0;
        _hbErrCoun := 0;

        fbServerCon
        (
            sSrvNetID     :=
            , nMode       := Tc2_TcpIp.CONNECT_MODE_ENABLEDBG
            , sRemoteHost := _sRemoteHost
            , nRemotePort := _serverPort
            , bEnable     := _bEnable
            , tReconnect  := reconnectTime
            , bBusy       => bBusy
            , bError      => bError
            , nErrId      => nErrId
            , hSocket     => hSocket
            , eState      => _eState
        );

        IF NOT fbServerCon.bBusy THEN
            IF NOT fbServerCon.bError THEN
                _n := _n + 1;

                IF _n >= 2 THEN
                    _n          := 0;
                    _bConnected := TRUE;

                    _msgFmtStr := 'Connection via TCP/IP established mit OmronRoboter! ';
                    Tc2_System.ADSLOGSTR
                    (
                        msgCtrlMask := Tc2_System.ADSLOG_MSGTYPE_WARN
                        , msgFmtStr := _msgFmtStr
                        , strArg    := ''
                    );

                    FaultID := 0;
                END_IF

                eStep := eCONNECTION_STATE_IDLE;
            ELSE
                _msgFmtStr := concat('fbServerCon geht nicht ', UDINT_TO_STRING(fbServerCon.nErrId));

                Tc2_System.ADSLOGSTR
                (
                    msgCtrlMask := Tc2_System.ADSLOG_MSGTYPE_WARN
                    , msgFmtStr := _msgFmtStr
                    , strArg    := ''
                );

                // Fehler, dass die Connection nicht zustande kommt fürs HMI
                // Lösung vermutlihc, Omron Comm-Programm muss neugestartet werden,
                // da ein Heartbeat FEhler vorliegt
                _bConnectedTrig(clk := _bConnected);
                FaultID := 10;
                eStep   := eCONNECTION_STATE_ERROR;
                _n      := 0;
            END_IF
        END_IF
    eCONNECTION_STATE_DATAEXCHANGE:
        _bDisconnect := NOT _bEnable OR _bDisconnect; //(kann aufs Hmi gelegt werden

        IF _bDisconnect AND NOT (fbSend.bBusy OR fbRceive.bBusy) THEN
            _bDisconnect := FALSE;
            eStep        := eCONNECTION_STATE_CLOSE_START;
        ELSE
            //Sender der Daten
            IF NOT (_bDisconnect OR fbSend.bBusy) THEN
                IF fbResponseTimer.q AND NOT fbRceive.bBusy THEN
                    fbSend(bExecute := FALSE);

                    fbSend
                    (
                        sSrvNetId  := sSrvNetId
                        , hSocket  := fbServerCon.hSocket
                        , cbLen    := cbLen
                        , pSrc     := ADR(msgSend.aTel)
                        , bExecute := TRUE
                        , tTimeout := tTimeout
                        , bBusy    => bBusy
                        , bError   => bError
                        , nErrId   => nErrId
                    );
                END_IF
            ELSE
                fbSend(bExecute := FALSE);

                IF fbSend.bError THEN
                    _msgFmtStr := concat('fbSend ', UDINT_TO_STRING(fbServerCon.nErrId));

                    Tc2_System.ADSLOGSTR
                    (
                        msgCtrlMask := Tc2_System.ADSLOG_MSGTYPE_WARN
                        , msgFmtStr := _msgFmtStr
                        , strArg    := ''
                    );
                END_IF
            END_IF

            //===================Recieve Data =================================
            IF NOT (_bDisconnect OR fbRceive.bBusy) THEN
                IF fbPollTimer.Q THEN
                    fbRceive(bExecute := FALSE);

                    fbRceive
                    (
                        sSrvNetId   := sSrvNetId
                        , hSocket   := fbServerCon.hSocket
                        , cbLen     := cbLen
                        , pDest     := ADR(msgRcv.aTel)
                        , bExecute  := TRUE
                        , tTimeout  := tTimeout
                        , bBusy     => bBusy
                        , bError    => bError
                        , nErrId    => nErrId
                        , nRecBytes =>
                    );

                    // CHekcehn des HEartbeats, ob Änderungen da sind
                    _hb := BYTE_TO_INT(msgRcv.stTel.myStats[3]);
                    fbRceive(nRecBytes => nRecBytes);

                    IF _hb = _hbOld THEN
                        fbTimeOut(in := TRUE);
                    ELSE
                        fbTimeOut(in := false);
                    END_IF

                    IF nRecBytes <> 0 THEN
                        IF _hb = _hbOld THEN
                            _hbErrCoun := _hbErrCoun + 1;

                            IF _hbErrCoun > 2 THEN
                                _ErrorCycle := _ErrorCycle + 1;
                            end_if
                        ELSIF _hb <> _hbOld OR _hb = 0 THEN
                            _hbErrCoun               := 0;
                            msgSend.stTel.myStats[3] := INT_TO_BYTE(_hb);
                        END_IF
                    END_IF

                    //===========================================================
                    //=========================================================
                    IF _hbErrCoun > hbError OR fbTimeOut.q THEN
                        _bDisconnect := TRUE;

                        //                        //                        mClearData();
                        FOR index := 1 TO UDINT_TO_UINT(cbLen) DO
                            msgRcv.aTel[index] := 0;
                        END_FOR

                        _msgFmtStr := 'HeartBeat Fehler, Verbindung verloren ';
                        Tc2_System.ADSLOGSTR
                        (
                            msgCtrlMask := Tc2_System.ADSLOG_MSGTYPE_WARN
                            , msgFmtStr := _msgFmtStr
                            , strArg    := ''
                        );
                    END_IF

                    _hbOld := _hb;
                END_IF
            ELSE
                fbRceive(bExecute := FALSE);

                IF NOT fbRceive.bError THEN
                    //watchdog von Omron, "HEartBeat"
                    //                    _msgSend.stTel.myStats[5] := _msgRcv.stTel.myStats[5];
                ELSE
                    _bDisconnect := TRUE;
                    _msgFmtStr   := concat('fbSocketRec ', UDINT_TO_STRING(fbRceive.nErrId));
                    Tc2_System.ADSLOGSTR
                    (
                        msgCtrlMask := Tc2_System.ADSLOG_MSGTYPE_WARN
                        , msgFmtStr := _msgFmtStr
                        , strArg    := ''
                    );
                END_IF
            END_IF
        END_IF
    eCONNECTION_STATE_CLOSE_START:
        Tc2_System.ADSLOGSTR
        (
            msgCtrlMask := Tc2_System.ADSLOG_MSGTYPE_WARN
            , msgFmtStr := 'Verbindung mit Omron wird geschlossen'
            , strArg    := ''
        );

        fbServerCon(bEnable := FALSE);
        fbTimeOut(in := FALSE);

        IF NOT fbServerCon.bBusy THEN
            _bConnected := FALSE;

            IF NOT fbServerCon.bError THEN
                eStep := eCONNECTION_STATE_IDLE;
            ELSE
                _msgFmtStr := concat('fbSocketClose ', UDINT_TO_STRING(fbServerCon.nErrId));

                Tc2_System.ADSLOGSTR
                (
                    msgCtrlMask := Tc2_System.ADSLOG_MSGTYPE_WARN
                    , msgFmtStr := _msgFmtStr
                    , strArg    := ''
                );

                eStep := eCONNECTION_STATE_ERROR;
            END_IF
        END_IF
    eCONNECTION_STATE_ERROR: (* Error step *)
        IF _bConnected THEN
            eStep := eCONNECTION_STATE_CLOSE_START;
        ELSE
            eStep := eCONNECTION_STATE_IDLE;
        END_IF
END_CASE
END_METHOD

END_FUNCTION_BLOCK

// ---- Test/CommunicationExtern Tests/CommunicationRoboterOmron_Test.TcPOU
FUNCTION_BLOCK CommunicationRoboterOmron_Test EXTENDS TcUnit.FB_TestSuite
VAR

END_VAR

SetOutputsExpectCorrespondingBits();

METHOD PRIVATE SetOutputsExpectCorrespondingBits
VAR_INST
    dut    : CommunicationRoboterOmron(sRemoteHost := '192.168.3.215', serverPort := 7000);
    itfDut : ICommunicationRoboterOmron ;


END_VAR
Test('SetOutputsExpectCorrespondingBits');
itfDut := dut;

dut.Run();
IF itfDut <> 0 THEN
    itfDut.Run();
    itfDut.ContactPrepared(TRUE);
    AssertTrue(dut.StatusCom.ContactPrepared, 'ContactPrepared muss true sein');

    itfDut.Reset(TRUE);
    AssertTrue(dut.StatusCom.Reset, 'Reset muss true sein');

end_if

TEST_FINISHED();
END_METHOD

END_FUNCTION_BLOCK

// ---- Test/SignalLights MachineStatus Tests/SignalLightsController_Test.TcPOU
FUNCTION_BLOCK INTERNAL SignalLightsController_Test EXTENDS TcUnit.FB_TestSuite IMPLEMENTS TcoCore.ITcoContext
VAR
    //Context for TcOpen
    _nfContext : TcoCore.TcoContextNfCompatibility;
END_VAR

SetModes_ExpectCorrLight();
SetMachineStatusOn_ExpectCorrLights();
SetIndivStatusOn_thenSetIndivOff();
SetMachineStatusOnAllThenOffAll();
SetDivStatus_ExpectPropsAccordingly();

PROPERTY Context : TcoCore.ITcoContext
GET
Context := This^._nfContext;
END_GET
END_PROPERTY

PROPERTY EndCycleCount : ULINT
GET
EndCycleCount := THIS^._nfContext._endCycleCount;
END_GET
END_PROPERTY

PROPERTY Environment : TcoCore.ITcoContextEnvironment
GET
Environment := THIS^._nfContext._settings;
END_GET
END_PROPERTY

PROPERTY Identity : ULINT
GET
Identity := THIS^._nfContext._Identity;
END_GET
END_PROPERTY

PROPERTY Logger : TcoCore.ITcoLogger
GET
Logger := THIS^._nfContext._logger;
END_GET
END_PROPERTY

PROPERTY RealTimeClock : TcoCore.ITcoRtc
GET
RealTimeClock := THIS^._nfContext._rtc;
END_GET
END_PROPERTY

METHOD PRIVATE SetDivStatus_ExpectPropsAccordingly
VAR_INST
    dut           : SignalLightsController(THIS^);
    itfDut        : ISignalLightsController;
    actualColor   : ColorsSignalLightsStatus;
    expectedColor : ColorsSignalLightsStatus;


    modesStatus : eMachineStatus;

END_VAR
TEST('SetDivStatus_ExpectPropsAccordingly');

//Arrange
itfDut := dut;

//Check before
AssertFalse(actualColor.Turquise, 'ColorOutput shall be off');
AssertFalse(actualColor.Blue, 'ColorOutput Blue shall be off');
AssertFalse(actualColor.Violet, 'ColorOuput Violet1 shall be off');
AssertFalse(actualColor.White, 'ColorOuput White shall be off');

//Blue
itfDut.SetMachineStatusOn(eMachineStatus.Blue);
actualColor := itfDut.GetColorsSignalLightMachineStatus;
AssertTrue(actualColor.Blue, 'ColorOutput Blue shall be On');
actualColor := itfDut.SetMachineStatusOff(eMachineStatus.Blue);
AssertFalse(actualColor.Blue, 'ColorOutput shall be off');

//Violet
actualColor := itfDut.SetMachineStatusOn(eMachineStatus.Violet);
AssertTrue(actualColor.Violet, 'ColorOutput Violet2 shall be On');
itfDut.SetMachineStatusOff(eMachineStatus.Violet);
actualColor := itfDut.GetColorsSignalLightMachineStatus;
AssertFalse(actualColor.Violet, 'ColorOutput Violet shall be Off');
AssertFalse(actualColor.Blue, 'ColorOutput shall be off');
actualColor := itfDut.SetMachineStatusOff(eMachineStatus.Violet);
AssertFalse(actualColor.Violet, 'ColorOutput shall be off');

//Turquise
actualColor := itfDut.SetMachineStatusOn(eMachineStatus.Turquise);
AssertTrue(actualColor.Turquise, 'ColorOutput Turquise shall be On');
AssertFalse(actualColor.White, 'ColorOutput shall be off');
AssertFalse(actualColor.Violet, 'ColorOutput shall be off');
AssertFalse(actualColor.Blue, 'ColorOutput shall be off');
actualColor := itfDut.SetMachineStatusOff(eMachineStatus.Turquise);
itfDut.SetMachineStatusOn(eMachineStatus.Turquise);
actualColor := itfDut.GetColorsSignalLightMachineStatus;
AssertTrue(actualColor.Turquise, 'ColorOutput Turquise shall be On');
itfDut.SetMachineStatusOff(eMachineStatus.Turquise);
actualColor := itfDut.GetColorsSignalLightMachineStatus;
AssertFalse(actualColor.Turquise, 'ColorOutput shall be off');
actualColor := itfDut.GetColorsSignalLightMachineStatus;
AssertFalse(actualColor.Turquise, 'ColorOutput shall be off');
//White
itfDut.SetMachineStatusOn(eMachineStatus.White);
actualColor := itfDut.GetColorsSignalLightMachineStatus;
AssertTrue(actualColor.White, 'ColorOutput White shall be On');
AssertFalse(actualColor.Turquise, 'ColorOutput shall be off');
actualColor := itfDut.SetMachineStatusOff(eMachineStatus.Violet);
AssertFalse(actualColor.Violet, 'ColorOutput shall be off');
AssertFalse(actualColor.Blue, 'ColorOutput shall be off');
actualColor := itfDut.SetMachineStatusOff(eMachineStatus.White);
AssertFalse(actualColor.White, 'ColorOutput shall be off');

{analysis -9}
TEST_FINISHED();
END_METHOD

METHOD PRIVATE SetIndivStatusOn_thenSetIndivOff
VAR_INST
    dut           : SignalLightsController(THIS^);
    itfDut        : ISignalLightsController;
    actualColor   : ColorsSignalLightsStatus;
    expectedColor : ColorsSignalLightsStatus;


    modesStatus : eMachineStatus;

END_VAR
TEST('SetIndivStatusOn_thenSetIndivOff');

//Arrange
itfDut := dut;

//Check before
AssertFalse(actualColor.Turquise, 'ColorOutput shall be off');
AssertFalse(actualColor.Blue, 'ColorOutput Blue shall be off');
AssertFalse(actualColor.Violet, 'ColorOuput Violet shall be off');
AssertFalse(actualColor.White, 'ColorOuput White shall be off');

//Blue
actualColor := itfDut.SetMachineStatusOn(eMachineStatus.Blue);
AssertTrue(actualColor.Blue, 'ColorOutput Blue shall be On');
 actualColor := itfDut.SetMachineStatusOff(eMachineStatus.Blue);
AssertFalse(actualColor.Blue, 'ColorOutput shall be off');

//Violet
actualColor :=itfDut.SetMachineStatusOn(eMachineStatus.Violet);
AssertTrue(actualColor.Violet, 'ColorOutput Violet shall be On');
AssertFalse(actualColor.Blue, 'ColorOutput shall be off');
actualColor :=itfDut.SetMachineStatusOff(eMachineStatus.Violet);
AssertFalse(actualColor.Violet, 'ColorOutput shall be off');

//Turquise
actualColor :=itfDut.SetMachineStatusOn(eMachineStatus.Turquise);
AssertTrue(actualColor.Turquise, 'ColorOutput Turquise shall be On');
AssertFalse(actualColor.White, 'ColorOutput shall be off');
AssertFalse(actualColor.Violet, 'ColorOutput shall be off');
AssertFalse(actualColor.Blue, 'ColorOutput shall be off');
actualColor :=itfDut.SetMachineStatusOff(eMachineStatus.Turquise);
actualColor :=itfDut.SetMachineStatusOn(eMachineStatus.Violet);
AssertTrue(actualColor.Violet, 'ColorOutput Violet shall be On');
AssertFalse(actualColor.Turquise, 'ColorOutput shall be off');

//White
actualColor :=itfDut.SetMachineStatusOn(eMachineStatus.White);
AssertTrue(actualColor.White, 'ColorOutput White shall be On');
AssertFalse(actualColor.Turquise, 'ColorOutput shall be off');
actualColor :=itfDut.SetMachineStatusOff(eMachineStatus.Violet);
AssertFalse(actualColor.Violet, 'ColorOutput shall be off');
AssertFalse(actualColor.Blue, 'ColorOutput shall be off');
actualColor :=itfDut.SetMachineStatusOff(eMachineStatus.White);
AssertFalse(actualColor.White , 'ColorOutput shall be off');

{analysis -9}
TEST_FINISHED();
END_METHOD

METHOD PRIVATE SetMachineStatusOn_ExpectCorrLights
VAR_INST
    dut           : SignalLightsController(THIS^);
    itfDut        : ISignalLightsController;
    actualColor   : ColorsSignalLightsStatus;
    expectedColor : ColorsSignalLightsStatus;
    modesStatus   : eMachineStatus;
END_VAR
TEST('SetMachineStatusOn_ExpectCorrLights');

//Arrange
itfDut := dut;

    modesStatus        := eMachineStatus.Blue;
    expectedColor.Blue := TRUE;

    // Act
    actualColor := itfDut.SetMachineStatusOn(modesStatus);

    // Assert
    AssertEquals
    (
        Expected  := expectedColor
        , Actual  := actualColor
        , Message := 'ColorOuput shall be BLUE'
    );

    //Act
    modesStatus := eMachineStatus.Turquise;
    actualColor := itfDut.SetMachineStatusOn(modesStatus);

    AssertTrue(actualColor.Turquise, 'ColorOutput shall be Turquise');
    AssertTrue(actualColor.Blue, 'ColorOutput Blue shall be still On');
    AssertFalse(actualColor.Violet, 'ColorOuput Violet shall be off');
    AssertFalse(actualColor.White, 'ColorOuput White shall be off');

     //Act
    modesStatus := eMachineStatus.Violet;
    actualColor := itfDut.SetMachineStatusOn(modesStatus);

    AssertTrue(actualColor.Turquise, 'ColorOutput shall be Turquise');
    AssertTrue(actualColor.Blue, 'ColorOutput Blue shall be still On');
    AssertTrue(actualColor.Violet, 'ColorOuput Violet shall be on');
    AssertFalse(actualColor.White, 'ColorOuput White shall be off');


         //Act
    modesStatus := eMachineStatus.White;
    actualColor := itfDut.SetMachineStatusOn(modesStatus);

    AssertTrue(actualColor.Turquise, 'ColorOutput shall be Turquise');
    AssertTrue(actualColor.Blue, 'ColorOutput Blue shall be still On');
    AssertTrue(actualColor.Violet, 'ColorOuput Violet shall be on');
    AssertTrue(actualColor.White, 'ColorOuput White shall be on');



         //Act
    modesStatus := eMachineStatus.All;
    actualColor := itfDut.SetMachineStatusOff(modesStatus);

    AssertFalse(actualColor.Turquise, 'ColorOutput shall be off');
    AssertFalse(actualColor.Blue, 'ColorOutput Blue shall be off');
    AssertFalse(actualColor.Violet, 'ColorOuput Violet shall be off');
    AssertFalse(actualColor.White, 'ColorOuput White shall be off');


{analysis -9}
TEST_FINISHED();
END_METHOD

METHOD PRIVATE SetMachineStatusOnAllThenOffAll
VAR_INST
    dut           : SignalLightsController(THIS^);
    itfDut        : ISignalLightsController;
    actualColor   : ColorsSignalLightsStatus;
    expectedColor : ColorsSignalLightsStatus;


    modesStatus : eMachineStatus;

END_VAR
TEST('SetMachineStatusOnAllThenOffAll');

//Arrange
itfDut := dut;

//Check before
AssertFalse(actualColor.Turquise, 'ColorOutput shall be off');
AssertFalse(actualColor.Blue, 'ColorOutput Blue shall be off');
AssertFalse(actualColor.Violet, 'ColorOuput Violet shall be off');
AssertFalse(actualColor.White, 'ColorOuput White shall be off');

//Act
actualColor := itfDut.SetMachineStatusOn(eMachineStatus.Blue);
actualColor := itfDut.SetMachineStatusOn(eMachineStatus.Turquise);
actualColor := itfDut.SetMachineStatusOn(eMachineStatus.Violet);
actualColor := itfDut.SetMachineStatusOn(eMachineStatus.White);

// Assert
AssertTrue(actualColor.Turquise, 'ColorOutput shall be Turquise');
AssertTrue(actualColor.Blue, 'ColorOutput Blue shall be still On');
AssertTrue(actualColor.Violet, 'ColorOuput Violet shall be On');
AssertTrue(actualColor.White, 'ColorOuput White shall be On');

//Act
actualColor := itfDut.SetMachineStatusOff(eMachineStatus.All);

//Check after
AssertFalse(actualColor.Turquise, 'ColorOutput shall be off');
AssertFalse(actualColor.Blue, 'ColorOutput Blue shall be off');
AssertFalse(actualColor.Violet, 'ColorOuput Violet shall be off');
AssertFalse(actualColor.White, 'ColorOuput White shall be off');

//setALll
actualColor := itfDut.SetMachineStatusOn(eMachineStatus.All);
// Assert
AssertTrue(actualColor.Turquise, 'ColorOutput shall be Turquise');
AssertTrue(actualColor.Blue, 'ColorOutput Blue shall be still On');
AssertTrue(actualColor.Violet, 'ColorOuput Violet shall be On');
AssertTrue(actualColor.White, 'ColorOuput White shall be On');
{analysis -9}
TEST_FINISHED();
END_METHOD

METHOD PRIVATE SetModes_ExpectCorrLight
VAR_INST

    dut           : SignalLightsController(THIS^);
    itfDut        : ISignalLightsController;
    actualColor   : ColorsSignalLightMachineModes;
    expectedColor : ColorsSignalLightMachineModes;

    blinkTime    : TIME := T#10MS;
    timer        : TON  := (pt := T#100MS);
    modesMachine : eMachineModes;
    state        : INT;

END_VAR
TEST('SetDifferentMachineModes_ExpectCorrespondingLightColor');

//Arrange
itfDut := dut;
itfDut.SetBlinkTime(blinktime, blinktime);

IF state = 0 THEN
    modesMachine        := eMachineModes.Automat;
    expectedColor.Green := TRUE;

    // Act
    actualColor := itfDut.SetMachineMode(modesMachine);

    // Assert
    AssertEquals
    (
        Expected  := expectedColor
        , Actual  := actualColor
        , Message := 'ColorOuput shall be Green'
    );

    //========================Idle=============================
    modesMachine         := eMachineModes.Idle;
    expectedColor.Green  := FALSE;
    expectedColor.Red    := FALSE;
    expectedColor.Yellow := FALSE;

    actualColor := itfDut.SetMachineMode(modesMachine);

    AssertEquals
    (
        Expected  := expectedColor
        , Actual  := actualColor
        , Message := 'ColorOuput shall be Off'
    );

    //========================Step=============================
    modesMachine         := eMachineModes.Step;
    expectedColor.Green  := TRUE;
    expectedColor.Red    := FALSE;
    expectedColor.Yellow := TRUE;

    actualColor := itfDut.SetMachineMode(modesMachine);

    AssertEquals
    (
        Expected  := expectedColor
        , Actual  := actualColor
        , Message := 'ColorOuput shall be GreenAndYellow'
    );

